LIN {X 0,Y 355.23,Z 732.233,A -85,B 0,C 180,E1 -13592.268,E2 -13592.268} C_VEL
LIN {X 0,Y 355.091,Z 732.252,A -85,B 0,C 180,E1 -13596.82,E2 -13596.82} C_VEL
LIN {X 0,Y 354.959,Z 732.267,A -85,B 0,C 180,E1 -13600.265,E2 -13600.265} C_VEL
LIN {X 0,Y 354.946,Z 732.27,A -85,B 0,C 180,E1 -13604.019,E2 -13604.019} C_VEL
LIN {X 0,Y 354.926,Z 732.273,A -85,B 0,C 180,E1 -13608.108,E2 -13608.108} C_VEL
LIN {X 0,Y 354.811,Z 732.288,A -85,B 0,C 180,E1 -13612.108,E2 -13612.108} C_VEL
LIN {X 0,Y 354.852,Z 732.28,A -85,B 0,C 180,E1 -13614.577,E2 -13614.577} C_VEL
LIN {X 0,Y 354.804,Z 732.288,A -85,B 0,C 180,E1 -13618.385,E2 -13618.385} C_VEL
LIN {X 0,Y 354.79,Z 732.291,A -85,B 0,C 180,E1 -13622.333,E2 -13622.333} C_VEL
LIN {X 0,Y 354.825,Z 732.285,A -85,B 0,C 180,E1 -13625.699,E2 -13625.699} C_VEL
LIN {X 0,Y 354.827,Z 732.283,A -85,B 0,C 180,E1 -13629.424,E2 -13629.424} C_VEL
LIN {X 0,Y 354.837,Z 732.433,A -85,B 0,C 180,E1 -13633.462,E2 -13633.462} C_VEL
LIN {X 0,Y 358.442,Z 744.759,A -85,B 0,C 180,E1 -13634.507,E2 -13634.507} C_VEL
LIN {X 0,Y 360.272,Z 752.132,A -85,B 0,C 180,E1 -13635.248,E2 -13635.248} C_VEL
LIN {X 0,Y 359.509,Z 762.827,A -85,B 0,C 180,E1 -13636.329,E2 -13636.329} C_VEL
LIN {X 0,Y 358.79,Z 772.72,A -85,B 0,C 180,E1 -13637.56,E2 -13637.56} C_VEL
LIN {X 0,Y 358.14,Z 780.809,A -85,B 0,C 180,E1 -13638.776,E2 -13638.776} C_VEL
LIN {X 0,Y 357.07,Z 784.926,A -85,B 0,C 180,E1 -13639.442,E2 -13639.442} C_VEL
LIN {X 0,Y 353.693,Z 791.298,A -85,B 0,C 180,E1 -13640.535,E2 -13640.535} C_VEL
LIN {X 0,Y 350.384,Z 797.153,A -85,B 0,C 180,E1 -13641.719,E2 -13641.719} C_VEL
LIN {X 0,Y 349.435,Z 800.343,A -85,B 0,C 180,E1 -13642.517,E2 -13642.517} C_VEL
LIN {X 0,Y 348.883,Z 806.047,A -85,B 0,C 180,E1 -13644.254,E2 -13644.254} C_VEL
LIN {X 0,Y 348.465,Z 811.428,A -85,B 0,C 180,E1 -13646.383,E2 -13646.383} C_VEL
LIN {X 0,Y 348.168,Z 814.944,A -85,B 0,C 180,E1 -13648.343,E2 -13648.343} C_VEL
LIN {X 0,Y 348.021,Z 817.216,A -85,B 0,C 180,E1 -13650.268,E2 -13650.268} C_VEL
LIN {X 0,Y 348.097,Z 818.5,A -85,B 0,C 180,E1 -13652.667,E2 -13652.667} C_VEL
LIN {X 0,Y 348.403,Z 818.075,A -85,B 0,C 180,E1 -13654.937,E2 -13654.937} C_VEL
LIN {X 0,Y 348.678,Z 817.181,A -85,B 0,C 180,E1 -13656.226,E2 -13656.226} C_VEL
LIN {X 0,Y 349.127,Z 815.318,A -85,B 0,C 180,E1 -13657.819,E2 -13657.819} C_VEL
LIN {X 0,Y 349.648,Z 812.667,A -85,B 0,C 180,E1 -13659.405,E2 -13659.405} C_VEL
LIN {X 0,Y 350.447,Z 808.387,A -85,B 0,C 180,E1 -13661.284,E2 -13661.284} C_VEL
LIN {X 0,Y 351.444,Z 802.773,A -85,B 0,C 180,E1 -13663.145,E2 -13663.145} C_VEL
LIN {X 0,Y 352.623,Z 795.572,A -85,B 0,C 180,E1 -13664.983,E2 -13664.983} C_VEL
LIN {X 0,Y 353.849,Z 787.076,A -85,B 0,C 180,E1 -13666.711,E2 -13666.711} C_VEL
LIN {X 0,Y 355.031,Z 778.224,A -85,B 0,C 180,E1 -13668.148,E2 -13668.148} C_VEL
LIN {X 0,Y 356.154,Z 768.152,A -85,B 0,C 180,E1 -13669.483,E2 -13669.483} C_VEL
LIN {X 0,Y 356.951,Z 758.725,A -85,B 0,C 180,E1 -13670.508,E2 -13670.508} C_VEL
LIN {X 0,Y 354.065,Z 748.897,A -85,B 0,C 180,E1 -13671.697,E2 -13671.697} C_VEL
LIN {X 0,Y 350.313,Z 738.899,A -85,B 0,C 180,E1 -13672.797,E2 -13672.797} C_VEL
LIN {X 0,Y 348.038,Z 733.135,A -85,B 0,C 180,E1 -13673.405,E2 -13673.405} C_VEL
LIN {X 0,Y 348.206,Z 733.113,A -85,B 0,C 180,E1 -13677.686,E2 -13677.686} C_VEL
LIN {X 0,Y 348.307,Z 733.1,A -85,B 0,C 180,E1 -13680,E2 -13680} C_VEL
LIN {X 0,Y 348.206,Z 733.106,A -85,B 0,C 180,E1 -13682.313,E2 -13682.313} C_VEL
LIN {X 0,Y 348.091,Z 733.123,A -85,B 0,C 180,E1 -13686.958,E2 -13686.958} C_VEL
LIN {X 0,Y 347.931,Z 733.145,A -85,B 0,C 180,E1 -13690.474,E2 -13690.474} C_VEL
LIN {X 0,Y 347.902,Z 733.146,A -85,B 0,C 180,E1 -13694.15,E2 -13694.15} C_VEL
LIN {X 0,Y 347.894,Z 733.145,A -85,B 0,C 180,E1 -13698.29,E2 -13698.29} C_VEL
LIN {X 0,Y 347.77,Z 733.16,A -85,B 0,C 180,E1 -13701.626,E2 -13701.626} C_VEL
LIN {X 0,Y 347.814,Z 733.16,A -85,B 0,C 180,E1 -13705.108,E2 -13705.108} C_VEL
LIN {X 0,Y 347.811,Z 733.161,A -85,B 0,C 180,E1 -13707.694,E2 -13707.694} C_VEL
LIN {X 0,Y 347.752,Z 733.168,A -85,B 0,C 180,E1 -13710.348,E2 -13710.348} C_VEL
LIN {X 0,Y 347.751,Z 733.169,A -85,B 0,C 180,E1 -13714.044,E2 -13714.044} C_VEL
LIN {X 0,Y 347.764,Z 733.169,A -85,B 0,C 180,E1 -13717.321,E2 -13717.321} C_VEL
LIN {X 0,Y 347.757,Z 733.181,A -85,B 0,C 180,E1 -13720.819,E2 -13720.819} C_VEL
LIN {X 0,Y 348.955,Z 738.713,A -85,B 0,C 180,E1 -13724.033,E2 -13724.033} C_VEL
LIN {X 0,Y 350.122,Z 744.422,A -85,B 0,C 180,E1 -13726.962,E2 -13726.962} C_VEL
LIN {X 0,Y 351.537,Z 751.508,A -85,B 0,C 180,E1 -13730.226,E2 -13730.226} C_VEL
LIN {X 0,Y 352.141,Z 756.915,A -85,B 0,C 180,E1 -13732.473,E2 -13732.473} C_VEL
LIN {X 0,Y 350.934,Z 766.228,A -85,B 0,C 180,E1 -13735.892,E2 -13735.892} C_VEL
LIN {X 0,Y 349.45,Z 779.49,A -85,B 0,C 180,E1 -13740.479,E2 -13740.479} C_VEL
LIN {X 0,Y 348.465,Z 791.054,A -85,B 0,C 180,E1 -13744.302,E2 -13744.302} C_VEL
LIN {X 0,Y 347.758,Z 802.825,A -85,B 0,C 180,E1 -13748.058,E2 -13748.058} C_VEL
LIN {X 0,Y 350.244,Z 818.097,A -85,B 0,C 180,E1 -13748.869,E2 -13748.869} C_VEL
LIN {X 0,Y 351.372,Z 830.122,A -85,B 0,C 180,E1 -13749.648,E2 -13749.648} C_VEL
LIN {X 0,Y 351.672,Z 841.978,A -85,B 0,C 180,E1 -13750.557,E2 -13750.557} C_VEL
LIN {X 0,Y 351.564,Z 853.712,A -85,B 0,C 180,E1 -13751.648,E2 -13751.648} C_VEL
LIN {X 0,Y 351.503,Z 860.57,A -85,B 0,C 180,E1 -13752.397,E2 -13752.397} C_VEL
LIN {X 0,Y 350.096,Z 871.051,A -85,B 0,C 180,E1 -13753.677,E2 -13753.677} C_VEL
LIN {X 0,Y 348.932,Z 881.081,A -85,B 0,C 180,E1 -13755.193,E2 -13755.193} C_VEL
LIN {X 0,Y 347.998,Z 890.121,A -85,B 0,C 180,E1 -13756.868,E2 -13756.868} C_VEL
LIN {X 0,Y 347.338,Z 897.875,A -85,B 0,C 180,E1 -13758.622,E2 -13758.622} C_VEL
LIN {X 0,Y 346.927,Z 905.128,A -85,B 0,C 180,E1 -13760.673,E2 -13760.673} C_VEL
LIN {X 0,Y 346.843,Z 910.019,A -85,B 0,C 180,E1 -13762.432,E2 -13762.432} C_VEL
LIN {X 0,Y 346.898,Z 913.8,A -85,B 0,C 180,E1 -13764.186,E2 -13764.186} C_VEL
LIN {X 0,Y 347.05,Z 915.739,A -85,B 0,C 180,E1 -13765.354,E2 -13765.354} C_VEL
LIN {X 0,Y 347.128,Z 917.246,A -85,B 0,C 180,E1 -13766.518,E2 -13766.518} C_VEL
LIN {X 0,Y 347.158,Z 918.314,A -85,B 0,C 180,E1 -13767.679,E2 -13767.679} C_VEL
LIN {X 0,Y 347.23,Z 918.922,A -85,B 0,C 180,E1 -13768.84,E2 -13768.84} C_VEL
LIN {X 0,Y 347.29,Z 919.114,A -85,B 0,C 180,E1 -13770,E2 -13770} C_VEL
LIN {X 0,Y 347.241,Z 918.877,A -85,B 0,C 180,E1 -13771.16,E2 -13771.16} C_VEL
LIN {X 0,Y 347.186,Z 918.212,A -85,B 0,C 180,E1 -13772.32,E2 -13772.32} C_VEL
LIN {X 0,Y 347.148,Z 917.076,A -85,B 0,C 180,E1 -13773.482,E2 -13773.482} C_VEL
LIN {X 0,Y 347.021,Z 914.544,A -85,B 0,C 180,E1 -13775.229,E2 -13775.229} C_VEL
LIN {X 0,Y 346.945,Z 910.936,A -85,B 0,C 180,E1 -13776.981,E2 -13776.981} C_VEL
LIN {X 0,Y 346.942,Z 906.157,A -85,B 0,C 180,E1 -13778.739,E2 -13778.739} C_VEL
LIN {X 0,Y 347.233,Z 898.965,A -85,B 0,C 180,E1 -13780.791,E2 -13780.791} C_VEL
LIN {X 0,Y 347.794,Z 891.13,A -85,B 0,C 180,E1 -13782.546,E2 -13782.546} C_VEL
LIN {X 0,Y 348.508,Z 883.149,A -85,B 0,C 180,E1 -13784.004,E2 -13784.004} C_VEL
LIN {X 0,Y 349.435,Z 873.459,A -85,B 0,C 180,E1 -13785.455,E2 -13785.455} C_VEL
LIN {X 0,Y 350.509,Z 862.791,A -85,B 0,C 180,E1 -13786.752,E2 -13786.752} C_VEL
LIN {X 0,Y 351.002,Z 857.17,A -85,B 0,C 180,E1 -13787.328,E2 -13787.328} C_VEL
LIN {X 0,Y 350.463,Z 844.972,A -85,B 0,C 180,E1 -13788.412,E2 -13788.412} C_VEL
LIN {X 0,Y 349.684,Z 831.983,A -85,B 0,C 180,E1 -13789.319,E2 -13789.319} C_VEL
LIN {X 0,Y 348.451,Z 818.444,A -85,B 0,C 180,E1 -13790.02,E2 -13790.02} C_VEL
LIN {X 0,Y 347.553,Z 809.771,A -85,B 0,C 180,E1 -13790.376,E2 -13790.376} C_VEL
LIN {X 0,Y 348.209,Z 799.166,A -85,B 0,C 180,E1 -13793.808,E2 -13793.808} C_VEL
LIN {X 0,Y 349.199,Z 787.298,A -85,B 0,C 180,E1 -13797.681,E2 -13797.681} C_VEL
LIN {X 0,Y 350.29,Z 775.966,A -85,B 0,C 180,E1 -13801.443,E2 -13801.443} C_VEL
LIN {X 0,Y 351.553,Z 765.595,A -85,B 0,C 180,E1 -13804.951,E2 -13804.951} C_VEL
LIN {X 0,Y 352.474,Z 758.03,A -85,B 0,C 180,E1 -13807.561,E2 -13807.561} C_VEL
LIN {X 0,Y 351.825,Z 753.478,A -85,B 0,C 180,E1 -13809.252,E2 -13809.252} C_VEL
LIN {X 0,Y 350.11,Z 744.683,A -85,B 0,C 180,E1 -13812.661,E2 -13812.661} C_VEL
LIN {X 0,Y 348.125,Z 735.001,A -85,B 0,C 180,E1 -13816.654,E2 -13816.654} C_VEL
LIN {X 0,Y 347.747,Z 733.17,A -85,B 0,C 180,E1 -13817.486,E2 -13817.486} C_VEL
LIN {X 0,Y 347.753,Z 733.168,A -85,B 0,C 180,E1 -13821.207,E2 -13821.207} C_VEL
LIN {X 0,Y 347.79,Z 733.161,A -85,B 0,C 180,E1 -13824.125,E2 -13824.125} C_VEL
LIN {X 0,Y 347.74,Z 733.169,A -85,B 0,C 180,E1 -13828.086,E2 -13828.086} C_VEL
LIN {X 0,Y 347.806,Z 733.157,A -85,B 0,C 180,E1 -13830.99,E2 -13830.99} C_VEL
LIN {X 0,Y 347.833,Z 733.157,A -85,B 0,C 180,E1 -13833.608,E2 -13833.608} C_VEL
LIN {X 0,Y 347.787,Z 733.164,A -85,B 0,C 180,E1 -13836.162,E2 -13836.162} C_VEL
LIN {X 0,Y 347.813,Z 733.161,A -85,B 0,C 180,E1 -13839.909,E2 -13839.909} C_VEL
LIN {X 0,Y 347.868,Z 733.154,A -85,B 0,C 180,E1 -13842.359,E2 -13842.359} C_VEL
LIN {X 0,Y 347.899,Z 733.149,A -85,B 0,C 180,E1 -13845.971,E2 -13845.971} C_VEL
LIN {X 0,Y 347.93,Z 733.142,A -85,B 0,C 180,E1 -13849.526,E2 -13849.526} C_VEL
LIN {X 0,Y 348.093,Z 733.123,A -85,B 0,C 180,E1 -13853.042,E2 -13853.042} C_VEL
LIN {X 0,Y 348.197,Z 733.109,A -85,B 0,C 180,E1 -13857.687,E2 -13857.687} C_VEL
LIN {X 0,Y 348.305,Z 733.096,A -85,B 0,C 180,E1 -13860,E2 -13860} C_VEL
LIN {X 0,Y 348.205,Z 733.11,A -85,B 0,C 180,E1 -13862.314,E2 -13862.314} C_VEL
LIN {X 0,Y 348.069,Z 733.13,A -85,B 0,C 180,E1 -13866.959,E2 -13866.959} C_VEL
LIN {X 0,Y 347.899,Z 733.148,A -85,B 0,C 180,E1 -13870.475,E2 -13870.475} C_VEL
LIN {X 0,Y 347.9,Z 733.146,A -85,B 0,C 180,E1 -13874.15,E2 -13874.15} C_VEL
LIN {X 0,Y 347.831,Z 733.155,A -85,B 0,C 180,E1 -13878.259,E2 -13878.259} C_VEL
LIN {X 0,Y 347.766,Z 733.166,A -85,B 0,C 180,E1 -13881.625,E2 -13881.625} C_VEL
LIN {X 0,Y 347.741,Z 733.17,A -85,B 0,C 180,E1 -13885.114,E2 -13885.114} C_VEL
LIN {X 0,Y 347.739,Z 733.17,A -85,B 0,C 180,E1 -13887.7,E2 -13887.7} C_VEL
LIN {X 0,Y 347.742,Z 733.166,A -85,B 0,C 180,E1 -13890.349,E2 -13890.349} C_VEL
LIN {X 0,Y 347.749,Z 733.167,A -85,B 0,C 180,E1 -13894.044,E2 -13894.044} C_VEL
LIN {X 0,Y 347.756,Z 733.167,A -85,B 0,C 180,E1 -13897.322,E2 -13897.322} C_VEL
LIN {X 0,Y 347.741,Z 733.17,A -85,B 0,C 180,E1 -13901.601,E2 -13901.601} C_VEL
LIN {X 0,Y 347.701,Z 733.171,A -85,B 0,C 180,E1 -13905.028,E2 -13905.028} C_VEL
LIN {X 0,Y 347.741,Z 733.169,A -85,B 0,C 180,E1 -13908.4,E2 -13908.4} C_VEL
LIN {X 0,Y 347.763,Z 733.168,A -85,B 0,C 180,E1 -13912.014,E2 -13912.014} C_VEL
LIN {X 0,Y 347.744,Z 733.166,A -85,B 0,C 180,E1 -13915.536,E2 -13915.536} C_VEL
LIN {X 0,Y 347.746,Z 733.17,A -85,B 0,C 180,E1 -13918.3,E2 -13918.3} C_VEL
LIN {X 0,Y 347.745,Z 733.166,A -85,B 0,C 180,E1 -13920.985,E2 -13920.985} C_VEL
LIN {X 0,Y 347.735,Z 733.167,A -85,B 0,C 180,E1 -13923.6,E2 -13923.6} C_VEL
LIN {X 0,Y 347.751,Z 733.168,A -85,B 0,C 180,E1 -13926.159,E2 -13926.159} C_VEL
LIN {X 0,Y 347.808,Z 733.158,A -85,B 0,C 180,E1 -13929.909,E2 -13929.909} C_VEL
LIN {X 0,Y 347.834,Z 733.154,A -85,B 0,C 180,E1 -13933.568,E2 -13933.568} C_VEL
LIN {X 0,Y 347.889,Z 733.15,A -85,B 0,C 180,E1 -13937.161,E2 -13937.161} C_VEL
LIN {X 0,Y 347.936,Z 733.146,A -85,B 0,C 180,E1 -13940.701,E2 -13940.701} C_VEL
LIN {X 0,Y 348.039,Z 733.129,A -85,B 0,C 180,E1 -13944.205,E2 -13944.205} C_VEL
LIN {X 0,Y 348.19,Z 733.111,A -85,B 0,C 180,E1 -13947.687,E2 -13947.687} C_VEL
LIN {X 0,Y 348.119,Z 733.124,A -85,B 0,C 180,E1 -13951.157,E2 -13951.157} C_VEL
LIN {X 0,Y 348.192,Z 733.11,A -85,B 0,C 180,E1 -13952.314,E2 -13952.314} C_VEL
LIN {X 0,Y 348.058,Z 733.129,A -85,B 0,C 180,E1 -13956.959,E2 -13956.959} C_VEL
LIN {X 0,Y 347.899,Z 733.146,A -85,B 0,C 180,E1 -13960.475,E2 -13960.475} C_VEL
LIN {X 0,Y 347.902,Z 733.147,A -85,B 0,C 180,E1 -13964.15,E2 -13964.15} C_VEL
LIN {X 0,Y 347.894,Z 733.147,A -85,B 0,C 180,E1 -13968.29,E2 -13968.29} C_VEL
LIN {X 0,Y 347.768,Z 733.167,A -85,B 0,C 180,E1 -13971.625,E2 -13971.625} C_VEL
LIN {X 0,Y 347.772,Z 733.162,A -85,B 0,C 180,E1 -13975.112,E2 -13975.112} C_VEL
LIN {X 0,Y 347.741,Z 733.169,A -85,B 0,C 180,E1 -13977.7,E2 -13977.7} C_VEL
LIN {X 0,Y 347.744,Z 733.168,A -85,B 0,C 180,E1 -13980.349,E2 -13980.349} C_VEL
LIN {X 0,Y 347.751,Z 733.169,A -85,B 0,C 180,E1 -13984.044,E2 -13984.044} C_VEL
LIN {X 0,Y 347.764,Z 733.162,A -85,B 0,C 180,E1 -13987.321,E2 -13987.321} C_VEL
LIN {X 0,Y 347.736,Z 733.172,A -85,B 0,C 180,E1 -13990.297,E2 -13990.297} C_VEL
LIN {X 0,Y 347.768,Z 733.163,A -85,B 0,C 180,E1 -13993.143,E2 -13993.143} C_VEL
LIN {X 0,Y 351.234,Z 745.101,A -85,B 0,C 180,E1 -13994.174,E2 -13994.174} C_VEL
LIN {X 0,Y 353.253,Z 752.532,A -85,B 0,C 180,E1 -13994.933,E2 -13994.933} C_VEL
LIN {X 0,Y 352.761,Z 762.272,A -85,B 0,C 180,E1 -13995.928,E2 -13995.928} C_VEL
LIN {X 0,Y 351.956,Z 772.866,A -85,B 0,C 180,E1 -13997.24,E2 -13997.24} C_VEL
LIN {X 0,Y 351.147,Z 782.229,A -85,B 0,C 180,E1 -13998.663,E2 -13998.663} C_VEL
LIN {X 0,Y 350.27,Z 791.601,A -85,B 0,C 180,E1 -14000.427,E2 -14000.427} C_VEL
LIN {X 0,Y 349.541,Z 799.315,A -85,B 0,C 180,E1 -14002.234,E2 -14002.234} C_VEL
LIN {X 0,Y 349.435,Z 800.343,A -85,B 0,C 180,E1 -14002.517,E2 -14002.517} C_VEL
LIN {X 0,Y 348.513,Z 803.347,A -85,B 0,C 180,E1 -14003.34,E2 -14003.34} C_VEL
LIN {X 0,Y 345.338,Z 807.953,A -85,B 0,C 180,E1 -14004.691,E2 -14004.691} C_VEL
LIN {X 0,Y 342.198,Z 811.889,A -85,B 0,C 180,E1 -14006.117,E2 -14006.117} C_VEL
LIN {X 0,Y 341.352,Z 813.811,A -85,B 0,C 180,E1 -14007.044,E2 -14007.044} C_VEL
LIN {X 0,Y 341.084,Z 816.896,A -85,B 0,C 180,E1 -14008.994,E2 -14008.994} C_VEL
LIN {X 0,Y 340.994,Z 818.317,A -85,B 0,C 180,E1 -14010.353,E2 -14010.353} C_VEL
LIN {X 0,Y 341.074,Z 819.469,A -85,B 0,C 180,E1 -14012.38,E2 -14012.38} C_VEL
LIN {X 0,Y 341.392,Z 819.241,A -85,B 0,C 180,E1 -14014.932,E2 -14014.932} C_VEL
LIN {X 0,Y 341.892,Z 817.661,A -85,B 0,C 180,E1 -14017.01,E2 -14017.01} C_VEL
LIN {X 0,Y 342.544,Z 815.006,A -85,B 0,C 180,E1 -14018.958,E2 -14018.958} C_VEL
LIN {X 0,Y 343.28,Z 811.201,A -85,B 0,C 180,E1 -14020.878,E2 -14020.878} C_VEL
LIN {X 0,Y 344.294,Z 806.037,A -85,B 0,C 180,E1 -14022.783,E2 -14022.783} C_VEL
LIN {X 0,Y 345.475,Z 799.43,A -85,B 0,C 180,E1 -14024.665,E2 -14024.665} C_VEL
LIN {X 0,Y 346.688,Z 792.011,A -85,B 0,C 180,E1 -14026.355,E2 -14026.355} C_VEL
LIN {X 0,Y 347.787,Z 784.502,A -85,B 0,C 180,E1 -14027.75,E2 -14027.75} C_VEL
LIN {X 0,Y 349.124,Z 774.386,A -85,B 0,C 180,E1 -14029.268,E2 -14029.268} C_VEL
LIN {X 0,Y 350.266,Z 763.595,A -85,B 0,C 180,E1 -14030.574,E2 -14030.574} C_VEL
LIN {X 0,Y 350.35,Z 760.277,A -85,B 0,C 180,E1 -14030.936,E2 -14030.936} C_VEL
LIN {X 0,Y 347.237,Z 749.774,A -85,B 0,C 180,E1 -14032.256,E2 -14032.256} C_VEL
LIN {X 0,Y 343.468,Z 739.901,A -85,B 0,C 180,E1 -14033.391,E2 -14033.391} C_VEL
LIN {X 0,Y 341.173,Z 734.849,A -85,B 0,C 180,E1 -14033.94,E2 -14033.94} C_VEL
LIN {X 0,Y 341.017,Z 734.004,A -85,B 0,C 180,E1 -14034.011,E2 -14034.011} C_VEL
LIN {X 0,Y 341.168,Z 733.989,A -85,B 0,C 180,E1 -14037.639,E2 -14037.639} C_VEL
LIN {X 0,Y 341.258,Z 733.978,A -85,B 0,C 180,E1 -14040,E2 -14040} C_VEL
LIN {X 0,Y 341.168,Z 733.982,A -85,B 0,C 180,E1 -14042.361,E2 -14042.361} C_VEL
LIN {X 0,Y 341.06,Z 733.999,A -85,B 0,C 180,E1 -14047.102,E2 -14047.102} C_VEL
LIN {X 0,Y 340.874,Z 734.023,A -85,B 0,C 180,E1 -14050.694,E2 -14050.694} C_VEL
LIN {X 0,Y 340.866,Z 734.021,A -85,B 0,C 180,E1 -14054.325,E2 -14054.325} C_VEL
LIN {X 0,Y 340.84,Z 734.024,A -85,B 0,C 180,E1 -14058.466,E2 -14058.466} C_VEL
LIN {X 0,Y 340.72,Z 734.039,A -85,B 0,C 180,E1 -14061.841,E2 -14061.841} C_VEL
LIN {X 0,Y 340.775,Z 734.037,A -85,B 0,C 180,E1 -14065.664,E2 -14065.664} C_VEL
LIN {X 0,Y 340.731,Z 734.04,A -85,B 0,C 180,E1 -14068.321,E2 -14068.321} C_VEL
LIN {X 0,Y 340.7,Z 734.043,A -85,B 0,C 180,E1 -14071.044,E2 -14071.044} C_VEL
LIN {X 0,Y 340.721,Z 734.043,A -85,B 0,C 180,E1 -14075.279,E2 -14075.279} C_VEL
LIN {X 0,Y 340.712,Z 734.049,A -85,B 0,C 180,E1 -14078.386,E2 -14078.386} C_VEL
LIN {X 0,Y 340.724,Z 734.107,A -85,B 0,C 180,E1 -14080.01,E2 -14080.01} C_VEL
LIN {X 0,Y 341.924,Z 739.628,A -85,B 0,C 180,E1 -14083.391,E2 -14083.391} C_VEL
LIN {X 0,Y 343.155,Z 745.722,A -85,B 0,C 180,E1 -14086.64,E2 -14086.64} C_VEL
LIN {X 0,Y 344.587,Z 752.85,A -85,B 0,C 180,E1 -14090.025,E2 -14090.025} C_VEL
LIN {X 0,Y 345.148,Z 756.489,A -85,B 0,C 180,E1 -14091.607,E2 -14091.607} C_VEL
LIN {X 0,Y 345.136,Z 758.878,A -85,B 0,C 180,E1 -14092.576,E2 -14092.576} C_VEL
LIN {X 0,Y 343.943,Z 767.473,A -85,B 0,C 180,E1 -14095.811,E2 -14095.811} C_VEL
LIN {X 0,Y 342.385,Z 780.646,A -85,B 0,C 180,E1 -14100.486,E2 -14100.486} C_VEL
LIN {X 0,Y 341.397,Z 792.174,A -85,B 0,C 180,E1 -14104.386,E2 -14104.386} C_VEL
LIN {X 0,Y 340.78,Z 801.684,A -85,B 0,C 180,E1 -14107.439,E2 -14107.439} C_VEL
LIN {X 0,Y 343.371,Z 816.716,A -85,B 0,C 180,E1 -14108.293,E2 -14108.293} C_VEL
LIN {X 0,Y 344.673,Z 829.763,A -85,B 0,C 180,E1 -14109.173,E2 -14109.173} C_VEL
LIN {X 0,Y 344.926,Z 842.378,A -85,B 0,C 180,E1 -14110.191,E2 -14110.191} C_VEL
LIN {X 0,Y 344.69,Z 854.862,A -85,B 0,C 180,E1 -14111.422,E2 -14111.422} C_VEL
LIN {X 0,Y 344.566,Z 861.431,A -85,B 0,C 180,E1 -14112.184,E2 -14112.184} C_VEL
LIN {X 0,Y 342.986,Z 872.499,A -85,B 0,C 180,E1 -14113.635,E2 -14113.635} C_VEL
LIN {X 0,Y 341.896,Z 881.316,A -85,B 0,C 180,E1 -14115.046,E2 -14115.046} C_VEL
LIN {X 0,Y 341.048,Z 889.379,A -85,B 0,C 180,E1 -14116.595,E2 -14116.595} C_VEL
LIN {X 0,Y 340.315,Z 897.076,A -85,B 0,C 180,E1 -14118.384,E2 -14118.384} C_VEL
LIN {X 0,Y 339.975,Z 902.361,A -85,B 0,C 180,E1 -14119.88,E2 -14119.88} C_VEL
LIN {X 0,Y 339.773,Z 907.59,A -85,B 0,C 180,E1 -14121.675,E2 -14121.675} C_VEL
LIN {X 0,Y 339.801,Z 910.959,A -85,B 0,C 180,E1 -14123.107,E2 -14123.107} C_VEL
LIN {X 0,Y 339.992,Z 914.762,A -85,B 0,C 180,E1 -14125.257,E2 -14125.257} C_VEL
LIN {X 0,Y 340.085,Z 916.259,A -85,B 0,C 180,E1 -14126.445,E2 -14126.445} C_VEL
LIN {X 0,Y 340.118,Z 917.295,A -85,B 0,C 180,E1 -14127.631,E2 -14127.631} C_VEL
LIN {X 0,Y 340.198,Z 917.888,A -85,B 0,C 180,E1 -14128.816,E2 -14128.816} C_VEL
LIN {X 0,Y 340.266,Z 918.068,A -85,B 0,C 180,E1 -14130,E2 -14130} C_VEL
LIN {X 0,Y 340.213,Z 917.818,A -85,B 0,C 180,E1 -14131.184,E2 -14131.184} C_VEL
LIN {X 0,Y 340.156,Z 917.115,A -85,B 0,C 180,E1 -14132.368,E2 -14132.368} C_VEL
LIN {X 0,Y 340.106,Z 915.956,A -85,B 0,C 180,E1 -14133.554,E2 -14133.554} C_VEL
LIN {X 0,Y 339.971,Z 913.383,A -85,B 0,C 180,E1 -14135.338,E2 -14135.338} C_VEL
LIN {X 0,Y 339.88,Z 909.726,A -85,B 0,C 180,E1 -14137.127,E2 -14137.127} C_VEL
LIN {X 0,Y 339.911,Z 904.901,A -85,B 0,C 180,E1 -14138.921,E2 -14138.921} C_VEL
LIN {X 0,Y 340.157,Z 898.783,A -85,B 0,C 180,E1 -14140.716,E2 -14140.716} C_VEL
LIN {X 0,Y 340.688,Z 891.179,A -85,B 0,C 180,E1 -14142.51,E2 -14142.51} C_VEL
LIN {X 0,Y 341.425,Z 883.438,A -85,B 0,C 180,E1 -14143.997,E2 -14143.997} C_VEL
LIN {X 0,Y 342.318,Z 874.012,A -85,B 0,C 180,E1 -14145.48,E2 -14145.48} C_VEL
LIN {X 0,Y 343.409,Z 863.657,A -85,B 0,C 180,E1 -14146.802,E2 -14146.802} C_VEL
LIN {X 0,Y 343.936,Z 856.845,A -85,B 0,C 180,E1 -14147.542,E2 -14147.542} C_VEL
LIN {X 0,Y 343.448,Z 844.854,A -85,B 0,C 180,E1 -14148.647,E2 -14148.647} C_VEL
LIN {X 0,Y 342.636,Z 831.043,A -85,B 0,C 180,E1 -14149.644,E2 -14149.644} C_VEL
LIN {X 0,Y 341.455,Z 817.895,A -85,B 0,C 180,E1 -14150.347,E2 -14150.347} C_VEL
LIN {X 0,Y 340.567,Z 808.849,A -85,B 0,C 180,E1 -14150.735,E2 -14150.735} C_VEL
LIN {X 0,Y 341.336,Z 796.876,A -85,B 0,C 180,E1 -14154.701,E2 -14154.701} C_VEL
LIN {X 0,Y 342.271,Z 786.494,A -85,B 0,C 180,E1 -14158.182,E2 -14158.182} C_VEL
LIN {X 0,Y 343.46,Z 774.864,A -85,B 0,C 180,E1 -14162.142,E2 -14162.142} C_VEL
LIN {X 0,Y 344.788,Z 764.543,A -85,B 0,C 180,E1 -14165.725,E2 -14165.725} C_VEL
LIN {X 0,Y 345.481,Z 759.219,A -85,B 0,C 180,E1 -14167.61,E2 -14167.61} C_VEL
LIN {X 0,Y 344.878,Z 754.873,A -85,B 0,C 180,E1 -14169.252,E2 -14169.252} C_VEL
LIN {X 0,Y 343.25,Z 746.62,A -85,B 0,C 180,E1 -14172.515,E2 -14172.515} C_VEL
LIN {X 0,Y 341.502,Z 738.052,A -85,B 0,C 180,E1 -14176.078,E2 -14176.078} C_VEL
LIN {X 0,Y 340.733,Z 734.042,A -85,B 0,C 180,E1 -14177.816,E2 -14177.816} C_VEL
LIN {X 0,Y 340.734,Z 734.043,A -85,B 0,C 180,E1 -14181.773,E2 -14181.773} C_VEL
LIN {X 0,Y 340.724,Z 734.044,A -85,B 0,C 180,E1 -14185.595,E2 -14185.595} C_VEL
LIN {X 0,Y 340.705,Z 734.042,A -85,B 0,C 180,E1 -14188.956,E2 -14188.956} C_VEL
LIN {X 0,Y 340.78,Z 734.034,A -85,B 0,C 180,E1 -14192.474,E2 -14192.474} C_VEL
LIN {X 0,Y 340.756,Z 734.038,A -85,B 0,C 180,E1 -14195.638,E2 -14195.638} C_VEL
LIN {X 0,Y 340.741,Z 734.038,A -85,B 0,C 180,E1 -14199.474,E2 -14199.474} C_VEL
LIN {X 0,Y 340.86,Z 734.027,A -85,B 0,C 180,E1 -14201.984,E2 -14201.984} C_VEL
LIN {X 0,Y 340.871,Z 734.022,A -85,B 0,C 180,E1 -14205.705,E2 -14205.705} C_VEL
LIN {X 0,Y 340.873,Z 734.021,A -85,B 0,C 180,E1 -14209.306,E2 -14209.306} C_VEL
LIN {X 0,Y 341.061,Z 734,A -85,B 0,C 180,E1 -14212.898,E2 -14212.898} C_VEL
LIN {X 0,Y 341.159,Z 733.985,A -85,B 0,C 180,E1 -14217.639,E2 -14217.639} C_VEL
LIN {X 0,Y 341.256,Z 733.974,A -85,B 0,C 180,E1 -14220,E2 -14220} C_VEL
LIN {X 0,Y 341.166,Z 733.987,A -85,B 0,C 180,E1 -14222.361,E2 -14222.361} C_VEL
LIN {X 0,Y 341.018,Z 734.007,A -85,B 0,C 180,E1 -14227.103,E2 -14227.103} C_VEL
LIN {X 0,Y 340.85,Z 734.028,A -85,B 0,C 180,E1 -14230.695,E2 -14230.695} C_VEL
LIN {X 0,Y 340.865,Z 734.023,A -85,B 0,C 180,E1 -14234.325,E2 -14234.325} C_VEL
LIN {X 0,Y 340.788,Z 734.032,A -85,B 0,C 180,E1 -14238.441,E2 -14238.441} C_VEL
LIN {X 0,Y 340.719,Z 734.042,A -85,B 0,C 180,E1 -14241.842,E2 -14241.842} C_VEL
LIN {X 0,Y 340.678,Z 734.049,A -85,B 0,C 180,E1 -14245.672,E2 -14245.672} C_VEL
LIN {X 0,Y 340.685,Z 734.045,A -85,B 0,C 180,E1 -14248.325,E2 -14248.325} C_VEL
LIN {X 0,Y 340.696,Z 734.045,A -85,B 0,C 180,E1 -14251.045,E2 -14251.045} C_VEL
LIN {X 0,Y 340.717,Z 734.043,A -85,B 0,C 180,E1 -14255.279,E2 -14255.279} C_VEL
LIN {X 0,Y 340.694,Z 734.044,A -85,B 0,C 180,E1 -14258.382,E2 -14258.382} C_VEL
LIN {X 0,Y 340.693,Z 734.048,A -85,B 0,C 180,E1 -14262.044,E2 -14262.044} C_VEL
LIN {X 0,Y 340.651,Z 734.052,A -85,B 0,C 180,E1 -14266.228,E2 -14266.228} C_VEL
LIN {X 0,Y 340.67,Z 734.047,A -85,B 0,C 180,E1 -14268.688,E2 -14268.688} C_VEL
LIN {X 0,Y 340.72,Z 734.043,A -85,B 0,C 180,E1 -14271.771,E2 -14271.771} C_VEL
LIN {X 0,Y 340.723,Z 734.041,A -85,B 0,C 180,E1 -14275.596,E2 -14275.596} C_VEL
LIN {X 0,Y 340.694,Z 734.044,A -85,B 0,C 180,E1 -14278.955,E2 -14278.955} C_VEL
LIN {X 0,Y 340.711,Z 734.042,A -85,B 0,C 180,E1 -14283.012,E2 -14283.012} C_VEL
LIN {X 0,Y 340.703,Z 734.045,A -85,B 0,C 180,E1 -14286.925,E2 -14286.925} C_VEL
LIN {X 0,Y 340.765,Z 734.04,A -85,B 0,C 180,E1 -14290.732,E2 -14290.732} C_VEL
LIN {X 0,Y 340.819,Z 734.031,A -85,B 0,C 180,E1 -14294.451,E2 -14294.451} C_VEL
LIN {X 0,Y 340.847,Z 734.025,A -85,B 0,C 180,E1 -14298.101,E2 -14298.101} C_VEL
LIN {X 0,Y 340.982,Z 734.008,A -85,B 0,C 180,E1 -14301.705,E2 -14301.705} C_VEL
LIN {X 0,Y 341.014,Z 734.004,A -85,B 0,C 180,E1 -14304.086,E2 -14304.086} C_VEL
LIN {X 0,Y 341.127,Z 733.991,A -85,B 0,C 180,E1 -14307.639,E2 -14307.639} C_VEL
LIN {X 0,Y 341.09,Z 733.999,A -85,B 0,C 180,E1 -14311.181,E2 -14311.181} C_VEL
LIN {X 0,Y 341.129,Z 733.989,A -85,B 0,C 180,E1 -14312.362,E2 -14312.362} C_VEL
LIN {X 0,Y 341.018,Z 734.004,A -85,B 0,C 180,E1 -14315.915,E2 -14315.915} C_VEL
LIN {X 0,Y 340.966,Z 734.009,A -85,B 0,C 180,E1 -14318.356,E2 -14318.356} C_VEL
LIN {X 0,Y 340.853,Z 734.026,A -85,B 0,C 180,E1 -14321.899,E2 -14321.899} C_VEL
LIN {X 0,Y 340.823,Z 734.033,A -85,B 0,C 180,E1 -14325.55,E2 -14325.55} C_VEL
LIN {X 0,Y 340.84,Z 734.025,A -85,B 0,C 180,E1 -14328.466,E2 -14328.466} C_VEL
LIN {X 0,Y 340.721,Z 734.046,A -85,B 0,C 180,E1 -14331.842,E2 -14331.842} C_VEL
LIN {X 0,Y 340.724,Z 734.044,A -85,B 0,C 180,E1 -14335.669,E2 -14335.669} C_VEL
LIN {X 0,Y 340.711,Z 734.044,A -85,B 0,C 180,E1 -14339.674,E2 -14339.674} C_VEL
LIN {X 0,Y 340.689,Z 734.046,A -85,B 0,C 180,E1 -14342.436,E2 -14342.436} C_VEL
LIN {X 0,Y 340.721,Z 734.04,A -85,B 0,C 180,E1 -14345.279,E2 -14345.279} C_VEL
LIN {X 0,Y 340.713,Z 734.045,A -85,B 0,C 180,E1 -14348.386,E2 -14348.386} C_VEL
LIN {X 0,Y 340.761,Z 734.038,A -85,B 0,C 180,E1 -14352.63,E2 -14352.63} C_VEL
LIN {X 0,Y 340.742,Z 734.04,A -85,B 0,C 180,E1 -14352.829,E2 -14352.829} C_VEL
LIN {X 0,Y 344.361,Z 746.61,A -85,B 0,C 180,E1 -14353.94,E2 -14353.94} C_VEL
LIN {X 0,Y 346.472,Z 754.427,A -85,B 0,C 180,E1 -14354.768,E2 -14354.768} C_VEL
LIN {X 0,Y 345.726,Z 765.186,A -85,B 0,C 180,E1 -14355.909,E2 -14355.909} C_VEL
LIN {X 0,Y 344.987,Z 774.871,A -85,B 0,C 180,E1 -14357.171,E2 -14357.171} C_VEL
LIN {X 0,Y 344.019,Z 785.198,A -85,B 0,C 180,E1 -14358.828,E2 -14358.828} C_VEL
LIN {X 0,Y 343.16,Z 794.057,A -85,B 0,C 180,E1 -14360.588,E2 -14360.588} C_VEL
LIN {X 0,Y 342.456,Z 801.226,A -85,B 0,C 180,E1 -14362.37,E2 -14362.37} C_VEL
LIN {X 0,Y 341.891,Z 806.952,A -85,B 0,C 180,E1 -14364.136,E2 -14364.136} C_VEL
LIN {X 0,Y 341.47,Z 812.236,A -85,B 0,C 180,E1 -14366.24,E2 -14366.24} C_VEL
LIN {X 0,Y 341.352,Z 813.811,A -85,B 0,C 180,E1 -14367.044,E2 -14367.044} C_VEL
LIN {X 0,Y 340.53,Z 815.559,A -85,B 0,C 180,E1 -14367.985,E2 -14367.985} C_VEL
LIN {X 0,Y 337.534,Z 818.043,A -85,B 0,C 180,E1 -14369.524,E2 -14369.524} C_VEL
LIN {X 0,Y 334.66,Z 819.863,A -85,B 0,C 180,E1 -14371.112,E2 -14371.112} C_VEL
LIN {X 0,Y 334.043,Z 820.431,A -85,B 0,C 180,E1 -14372.113,E2 -14372.113} C_VEL
LIN {X 0,Y 334.205,Z 820.699,A -85,B 0,C 180,E1 -14373.793,E2 -14373.793} C_VEL
LIN {X 0,Y 334.425,Z 820.306,A -85,B 0,C 180,E1 -14375.146,E2 -14375.146} C_VEL
LIN {X 0,Y 335.019,Z 818.596,A -85,B 0,C 180,E1 -14377.374,E2 -14377.374} C_VEL
LIN {X 0,Y 335.646,Z 816.186,A -85,B 0,C 180,E1 -14379.148,E2 -14379.148} C_VEL
LIN {X 0,Y 336.422,Z 812.421,A -85,B 0,C 180,E1 -14381.107,E2 -14381.107} C_VEL
LIN {X 0,Y 337.616,Z 806.705,A -85,B 0,C 180,E1 -14383.25,E2 -14383.25} C_VEL
LIN {X 0,Y 338.957,Z 799.58,A -85,B 0,C 180,E1 -14385.286,E2 -14385.286} C_VEL
LIN {X 0,Y 340.191,Z 792.572,A -85,B 0,C 180,E1 -14386.865,E2 -14386.865} C_VEL
LIN {X 0,Y 341.494,Z 784.065,A -85,B 0,C 180,E1 -14388.424,E2 -14388.424} C_VEL
LIN {X 0,Y 342.847,Z 774.065,A -85,B 0,C 180,E1 -14389.909,E2 -14389.909} C_VEL
LIN {X 0,Y 343.961,Z 763.803,A -85,B 0,C 180,E1 -14391.148,E2 -14391.148} C_VEL
LIN {X 0,Y 343.601,Z 761.252,A -85,B 0,C 180,E1 -14391.472,E2 -14391.472} C_VEL
LIN {X 0,Y 340.343,Z 750.418,A -85,B 0,C 180,E1 -14392.883,E2 -14392.883} C_VEL
LIN {X 0,Y 336.591,Z 741.093,A -85,B 0,C 180,E1 -14394.007,E2 -14394.007} C_VEL
LIN {X 0,Y 334.012,Z 735.653,A -85,B 0,C 180,E1 -14394.642,E2 -14394.642} C_VEL
LIN {X 0,Y 333.86,Z 734.895,A -85,B 0,C 180,E1 -14394.716,E2 -14394.716} C_VEL
LIN {X 0,Y 334.105,Z 734.869,A -85,B 0,C 180,E1 -14397.589,E2 -14397.589} C_VEL
LIN {X 0,Y 334.21,Z 734.856,A -85,B 0,C 180,E1 -14400,E2 -14400} C_VEL
LIN {X 0,Y 334.105,Z 734.862,A -85,B 0,C 180,E1 -14402.411,E2 -14402.411} C_VEL
LIN {X 0,Y 334.016,Z 734.872,A -85,B 0,C 180,E1 -14406.039,E2 -14406.039} C_VEL
LIN {X 0,Y 333.962,Z 734.878,A -85,B 0,C 180,E1 -14408.471,E2 -14408.471} C_VEL
LIN {X 0,Y 333.794,Z 734.9,A -85,B 0,C 180,E1 -14412.154,E2 -14412.154} C_VEL
LIN {X 0,Y 333.781,Z 734.903,A -85,B 0,C 180,E1 -14415.886,E2 -14415.886} C_VEL
LIN {X 0,Y 333.799,Z 734.901,A -85,B 0,C 180,E1 -14418.655,E2 -14418.655} C_VEL
LIN {X 0,Y 333.66,Z 734.924,A -85,B 0,C 180,E1 -14422.28,E2 -14422.28} C_VEL
LIN {X 0,Y 333.737,Z 734.909,A -85,B 0,C 180,E1 -14426.246,E2 -14426.246} C_VEL
LIN {X 0,Y 333.693,Z 734.915,A -85,B 0,C 180,E1 -14428.974,E2 -14428.974} C_VEL
LIN {X 0,Y 333.648,Z 734.924,A -85,B 0,C 180,E1 -14432.587,E2 -14432.587} C_VEL
LIN {X 0,Y 333.679,Z 734.926,A -85,B 0,C 180,E1 -14436.139,E2 -14436.139} C_VEL
LIN {X 0,Y 333.667,Z 735.104,A -85,B 0,C 180,E1 -14439.19,E2 -14439.19} C_VEL
LIN {X 0,Y 334.927,Z 740.587,A -85,B 0,C 180,E1 -14442.74,E2 -14442.74} C_VEL
LIN {X 0,Y 336.245,Z 747.17,A -85,B 0,C 180,E1 -14446.389,E2 -14446.389} C_VEL
LIN {X 0,Y 337.641,Z 754.183,A -85,B 0,C 180,E1 -14449.814,E2 -14449.814} C_VEL
LIN {X 0,Y 338.269,Z 759.458,A -85,B 0,C 180,E1 -14452.139,E2 -14452.139} C_VEL
LIN {X 0,Y 337.2,Z 766.879,A -85,B 0,C 180,E1 -14455.029,E2 -14455.029} C_VEL
LIN {X 0,Y 335.9,Z 776.168,A -85,B 0,C 180,E1 -14458.461,E2 -14458.461} C_VEL
LIN {X 0,Y 334.901,Z 786.533,A -85,B 0,C 180,E1 -14462.143,E2 -14462.143} C_VEL
LIN {X 0,Y 334.013,Z 797.145,A -85,B 0,C 180,E1 -14465.776,E2 -14465.776} C_VEL
LIN {X 0,Y 333.825,Z 800.305,A -85,B 0,C 180,E1 -14466.77,E2 -14466.77} C_VEL
LIN {X 0,Y 336.377,Z 814.35,A -85,B 0,C 180,E1 -14467.605,E2 -14467.605} C_VEL
LIN {X 0,Y 337.906,Z 828.047,A -85,B 0,C 180,E1 -14468.574,E2 -14468.574} C_VEL
LIN {X 0,Y 338.224,Z 841.628,A -85,B 0,C 180,E1 -14469.707,E2 -14469.707} C_VEL
LIN {X 0,Y 337.915,Z 853.273,A -85,B 0,C 180,E1 -14470.878,E2 -14470.878} C_VEL
LIN {X 0,Y 337.636,Z 862.278,A -85,B 0,C 180,E1 -14471.963,E2 -14471.963} C_VEL
LIN {X 0,Y 336.122,Z 871.993,A -85,B 0,C 180,E1 -14473.291,E2 -14473.291} C_VEL
LIN {X 0,Y 334.841,Z 881.661,A -85,B 0,C 180,E1 -14474.906,E2 -14474.906} C_VEL
LIN {X 0,Y 333.902,Z 890.015,A -85,B 0,C 180,E1 -14476.613,E2 -14476.613} C_VEL
LIN {X 0,Y 333.093,Z 898.459,A -85,B 0,C 180,E1 -14478.745,E2 -14478.745} C_VEL
LIN {X 0,Y 332.742,Z 905.106,A -85,B 0,C 180,E1 -14480.885,E2 -14480.885} C_VEL
LIN {X 0,Y 332.721,Z 910.317,A -85,B 0,C 180,E1 -14483.107,E2 -14483.107} C_VEL
LIN {X 0,Y 332.915,Z 913.787,A -85,B 0,C 180,E1 -14485.156,E2 -14485.156} C_VEL
LIN {X 0,Y 333.042,Z 915.272,A -85,B 0,C 180,E1 -14486.37,E2 -14486.37} C_VEL
LIN {X 0,Y 333.078,Z 916.276,A -85,B 0,C 180,E1 -14487.581,E2 -14487.581} C_VEL
LIN {X 0,Y 333.165,Z 916.859,A -85,B 0,C 180,E1 -14488.791,E2 -14488.791} C_VEL
LIN {X 0,Y 333.242,Z 917.027,A -85,B 0,C 180,E1 -14490,E2 -14490} C_VEL
LIN {X 0,Y 333.185,Z 916.757,A -85,B 0,C 180,E1 -14491.209,E2 -14491.209} C_VEL
LIN {X 0,Y 333.124,Z 916.016,A -85,B 0,C 180,E1 -14492.418,E2 -14492.418} C_VEL
LIN {X 0,Y 333.064,Z 914.84,A -85,B 0,C 180,E1 -14493.629,E2 -14493.629} C_VEL
LIN {X 0,Y 332.924,Z 912.224,A -85,B 0,C 180,E1 -14495.451,E2 -14495.451} C_VEL
LIN {X 0,Y 332.83,Z 908.52,A -85,B 0,C 180,E1 -14497.279,E2 -14497.279} C_VEL
LIN {X 0,Y 332.86,Z 903.644,A -85,B 0,C 180,E1 -14499.111,E2 -14499.111} C_VEL
LIN {X 0,Y 333.123,Z 897.471,A -85,B 0,C 180,E1 -14500.945,E2 -14500.945} C_VEL
LIN {X 0,Y 333.697,Z 889.797,A -85,B 0,C 180,E1 -14502.776,E2 -14502.776} C_VEL
LIN {X 0,Y 334.392,Z 881.95,A -85,B 0,C 180,E1 -14504.297,E2 -14504.297} C_VEL
LIN {X 0,Y 335.563,Z 871.386,A -85,B 0,C 180,E1 -14505.955,E2 -14505.955} C_VEL
LIN {X 0,Y 336.551,Z 861.98,A -85,B 0,C 180,E1 -14507.155,E2 -14507.155} C_VEL
LIN {X 0,Y 336.849,Z 854.973,A -85,B 0,C 180,E1 -14507.923,E2 -14507.923} C_VEL
LIN {X 0,Y 336.368,Z 842.767,A -85,B 0,C 180,E1 -14509.054,E2 -14509.054} C_VEL
LIN {X 0,Y 335.525,Z 829.149,A -85,B 0,C 180,E1 -14510.043,E2 -14510.043} C_VEL
LIN {X 0,Y 334.222,Z 815.094,A -85,B 0,C 180,E1 -14510.784,E2 -14510.784} C_VEL
LIN {X 0,Y 333.533,Z 807.992,A -85,B 0,C 180,E1 -14511.068,E2 -14511.068} C_VEL
LIN {X 0,Y 334.39,Z 795.433,A -85,B 0,C 180,E1 -14515.345,E2 -14515.345} C_VEL
LIN {X 0,Y 335.37,Z 785.344,A -85,B 0,C 180,E1 -14518.815,E2 -14518.815} C_VEL
LIN {X 0,Y 336.668,Z 773.737,A -85,B 0,C 180,E1 -14522.871,E2 -14522.871} C_VEL
LIN {X 0,Y 337.994,Z 763.987,A -85,B 0,C 180,E1 -14526.344,E2 -14526.344} C_VEL
LIN {X 0,Y 338.462,Z 759.697,A -85,B 0,C 180,E1 -14527.903,E2 -14527.903} C_VEL
LIN {X 0,Y 337.179,Z 752.397,A -85,B 0,C 180,E1 -14530.777,E2 -14530.777} C_VEL
LIN {X 0,Y 335.328,Z 743.269,A -85,B 0,C 180,E1 -14534.554,E2 -14534.554} C_VEL
LIN {X 0,Y 333.671,Z 734.923,A -85,B 0,C 180,E1 -14538.233,E2 -14538.233} C_VEL
LIN {X 0,Y 333.653,Z 734.921,A -85,B 0,C 180,E1 -14542.349,E2 -14542.349} C_VEL
LIN {X 0,Y 333.675,Z 734.92,A -85,B 0,C 180,E1 -14545.341,E2 -14545.341} C_VEL
LIN {X 0,Y 333.704,Z 734.919,A -85,B 0,C 180,E1 -14549.71,E2 -14549.71} C_VEL
LIN {X 0,Y 333.745,Z 734.91,A -85,B 0,C 180,E1 -14552.401,E2 -14552.401} C_VEL
LIN {X 0,Y 333.727,Z 734.911,A -85,B 0,C 180,E1 -14555.091,E2 -14555.091} C_VEL
LIN {X 0,Y 333.678,Z 734.917,A -85,B 0,C 180,E1 -14559.019,E2 -14559.019} C_VEL
LIN {X 0,Y 333.796,Z 734.904,A -85,B 0,C 180,E1 -14561.59,E2 -14561.59} C_VEL
LIN {X 0,Y 333.81,Z 734.901,A -85,B 0,C 180,E1 -14565.577,E2 -14565.577} C_VEL
LIN {X 0,Y 333.836,Z 734.898,A -85,B 0,C 180,E1 -14569.078,E2 -14569.078} C_VEL
LIN {X 0,Y 334.008,Z 734.88,A -85,B 0,C 180,E1 -14572.747,E2 -14572.747} C_VEL
LIN {X 0,Y 333.8,Z 734.903,A -85,B 0,C 180,E1 -14575.169,E2 -14575.169} C_VEL
LIN {X 0,Y 334.096,Z 734.865,A -85,B 0,C 180,E1 -14577.589,E2 -14577.589} C_VEL
LIN {X 0,Y 334.208,Z 734.852,A -85,B 0,C 180,E1 -14580,E2 -14580} C_VEL
LIN {X 0,Y 334.103,Z 734.867,A -85,B 0,C 180,E1 -14582.411,E2 -14582.411} C_VEL
LIN {X 0,Y 333.97,Z 734.88,A -85,B 0,C 180,E1 -14586.52,E2 -14586.52} C_VEL
LIN {X 0,Y 333.822,Z 734.9,A -85,B 0,C 180,E1 -14589.696,E2 -14589.696} C_VEL
LIN {X 0,Y 333.799,Z 734.905,A -85,B 0,C 180,E1 -14593.392,E2 -14593.392} C_VEL
LIN {X 0,Y 333.722,Z 734.918,A -85,B 0,C 180,E1 -14597.148,E2 -14597.148} C_VEL
LIN {X 0,Y 333.691,Z 734.917,A -85,B 0,C 180,E1 -14599.693,E2 -14599.693} C_VEL
LIN {X 0,Y 333.644,Z 734.925,A -85,B 0,C 180,E1 -14603.592,E2 -14603.592} C_VEL
LIN {X 0,Y 333.67,Z 734.923,A -85,B 0,C 180,E1 -14607.606,E2 -14607.606} C_VEL
LIN {X 0,Y 333.659,Z 734.92,A -85,B 0,C 180,E1 -14610.366,E2 -14610.366} C_VEL
LIN {X 0,Y 333.638,Z 734.925,A -85,B 0,C 180,E1 -14613.209,E2 -14613.209} C_VEL
LIN {X 0,Y 333.675,Z 734.919,A -85,B 0,C 180,E1 -14616.14,E2 -14616.14} C_VEL
LIN {X 0,Y 333.603,Z 734.928,A -85,B 0,C 180,E1 -14619.199,E2 -14619.199} C_VEL
LIN {X 0,Y 333.628,Z 734.924,A -85,B 0,C 180,E1 -14622.499,E2 -14622.499} C_VEL
LIN {X 0,Y 333.595,Z 734.933,A -85,B 0,C 180,E1 -14625.955,E2 -14625.955} C_VEL
LIN {X 0,Y 333.603,Z 734.927,A -85,B 0,C 180,E1 -14629.325,E2 -14629.325} C_VEL
LIN {X 0,Y 333.663,Z 734.919,A -85,B 0,C 180,E1 -14633.169,E2 -14633.169} C_VEL
LIN {X 0,Y 333.674,Z 734.918,A -85,B 0,C 180,E1 -14635.341,E2 -14635.341} C_VEL
LIN {X 0,Y 333.631,Z 734.929,A -85,B 0,C 180,E1 -14638.222,E2 -14638.222} C_VEL
LIN {X 0,Y 333.631,Z 734.924,A -85,B 0,C 180,E1 -14641.02,E2 -14641.02} C_VEL
LIN {X 0,Y 333.659,Z 734.922,A -85,B 0,C 180,E1 -14644.922,E2 -14644.922} C_VEL
LIN {X 0,Y 333.668,Z 734.92,A -85,B 0,C 180,E1 -14649.018,E2 -14649.018} C_VEL
LIN {X 0,Y 333.744,Z 734.909,A -85,B 0,C 180,E1 -14651.587,E2 -14651.587} C_VEL
LIN {X 0,Y 333.811,Z 734.901,A -85,B 0,C 180,E1 -14655.577,E2 -14655.577} C_VEL
LIN {X 0,Y 333.816,Z 734.904,A -85,B 0,C 180,E1 -14659.078,E2 -14659.078} C_VEL
LIN {X 0,Y 333.958,Z 734.886,A -85,B 0,C 180,E1 -14662.746,E2 -14662.746} C_VEL
LIN {X 0,Y 333.778,Z 734.91,A -85,B 0,C 180,E1 -14665.169,E2 -14665.169} C_VEL
LIN {X 0,Y 334.067,Z 734.87,A -85,B 0,C 180,E1 -14667.589,E2 -14667.589} C_VEL
LIN {X 0,Y 334.061,Z 734.875,A -85,B 0,C 180,E1 -14671.206,E2 -14671.206} C_VEL
LIN {X 0,Y 334.069,Z 734.869,A -85,B 0,C 180,E1 -14672.412,E2 -14672.412} C_VEL
LIN {X 0,Y 333.992,Z 734.879,A -85,B 0,C 180,E1 -14676.04,E2 -14676.04} C_VEL
LIN {X 0,Y 333.823,Z 734.903,A -85,B 0,C 180,E1 -14679.696,E2 -14679.696} C_VEL
LIN {X 0,Y 333.8,Z 734.907,A -85,B 0,C 180,E1 -14683.391,E2 -14683.391} C_VEL
LIN {X 0,Y 333.75,Z 734.91,A -85,B 0,C 180,E1 -14687.146,E2 -14687.146} C_VEL
LIN {X 0,Y 333.735,Z 734.916,A -85,B 0,C 180,E1 -14689.691,E2 -14689.691} C_VEL
LIN {X 0,Y 333.66,Z 734.923,A -85,B 0,C 180,E1 -14693.591,E2 -14693.591} C_VEL
LIN {X 0,Y 333.66,Z 734.922,A -85,B 0,C 180,E1 -14696.253,E2 -14696.253} C_VEL
LIN {X 0,Y 333.665,Z 734.922,A -85,B 0,C 180,E1 -14700.278,E2 -14700.278} C_VEL
LIN {X 0,Y 333.64,Z 734.922,A -85,B 0,C 180,E1 -14703.208,E2 -14703.208} C_VEL
LIN {X 0,Y 333.679,Z 734.923,A -85,B 0,C 180,E1 -14706.139,E2 -14706.139} C_VEL
LIN {X 0,Y 333.65,Z 734.92,A -85,B 0,C 180,E1 -14709.192,E2 -14709.192} C_VEL
LIN {X 0,Y 333.721,Z 734.916,A -85,B 0,C 180,E1 -14712.491,E2 -14712.491} C_VEL
LIN {X 0,Y 337.361,Z 747.471,A -85,B 0,C 180,E1 -14713.635,E2 -14713.635} C_VEL
LIN {X 0,Y 339.539,Z 755.639,A -85,B 0,C 180,E1 -14714.521,E2 -14714.521} C_VEL
LIN {X 0,Y 338.878,Z 765.769,A -85,B 0,C 180,E1 -14715.619,E2 -14715.619} C_VEL
LIN {X 0,Y 338.001,Z 776.704,A -85,B 0,C 180,E1 -14717.08,E2 -14717.08} C_VEL
LIN {X 0,Y 337.083,Z 786.192,A -85,B 0,C 180,E1 -14718.641,E2 -14718.641} C_VEL
LIN {X 0,Y 336.253,Z 794.413,A -85,B 0,C 180,E1 -14720.291,E2 -14720.291} C_VEL
LIN {X 0,Y 335.474,Z 802.085,A -85,B 0,C 180,E1 -14722.209,E2 -14722.209} C_VEL
LIN {X 0,Y 334.897,Z 807.847,A -85,B 0,C 180,E1 -14724.013,E2 -14724.013} C_VEL
LIN {X 0,Y 334.448,Z 813.17,A -85,B 0,C 180,E1 -14726.16,E2 -14726.16} C_VEL
LIN {X 0,Y 334.135,Z 816.927,A -85,B 0,C 180,E1 -14728.275,E2 -14728.275} C_VEL
LIN {X 0,Y 334.003,Z 818.675,A -85,B 0,C 180,E1 -14729.668,E2 -14729.668} C_VEL
LIN {X 0,Y 333.976,Z 819.886,A -85,B 0,C 180,E1 -14731.053,E2 -14731.053} C_VEL
LIN {X 0,Y 334.043,Z 820.431,A -85,B 0,C 180,E1 -14732.113,E2 -14732.113} C_VEL
LIN {X 0,Y 333.481,Z 820.778,A -85,B 0,C 180,E1 -14733.122,E2 -14733.122} C_VEL
LIN {X 0,Y 330.908,Z 821.1,A -85,B 0,C 180,E1 -14734.773,E2 -14734.773} C_VEL
LIN {X 0,Y 328.443,Z 820.675,A -85,B 0,C 180,E1 -14736.441,E2 -14736.441} C_VEL
LIN {X 0,Y 328.056,Z 819.801,A -85,B 0,C 180,E1 -14737.459,E2 -14737.459} C_VEL
LIN {X 0,Y 328.746,Z 817.392,A -85,B 0,C 180,E1 -14739.345,E2 -14739.345} C_VEL
LIN {X 0,Y 329.582,Z 813.677,A -85,B 0,C 180,E1 -14741.345,E2 -14741.345} C_VEL
LIN {X 0,Y 330.836,Z 808.015,A -85,B 0,C 180,E1 -14743.533,E2 -14743.533} C_VEL
LIN {X 0,Y 332.24,Z 800.998,A -85,B 0,C 180,E1 -14745.592,E2 -14745.592} C_VEL
LIN {X 0,Y 333.556,Z 793.98,A -85,B 0,C 180,E1 -14747.218,E2 -14747.218} C_VEL
LIN {X 0,Y 334.936,Z 785.58,A -85,B 0,C 180,E1 -14748.808,E2 -14748.808} C_VEL
LIN {X 0,Y 336.226,Z 776.745,A -85,B 0,C 180,E1 -14750.176,E2 -14750.176} C_VEL
LIN {X 0,Y 337.625,Z 765.201,A -85,B 0,C 180,E1 -14751.621,E2 -14751.621} C_VEL
LIN {X 0,Y 334.967,Z 755.721,A -85,B 0,C 180,E1 -14752.938,E2 -14752.938} C_VEL
LIN {X 0,Y 331.436,Z 746.12,A -85,B 0,C 180,E1 -14754.188,E2 -14754.188} C_VEL
LIN {X 0,Y 328.076,Z 739.094,A -85,B 0,C 180,E1 -14755.084,E2 -14755.084} C_VEL
LIN {X 0,Y 326.812,Z 736.178,A -85,B 0,C 180,E1 -14755.413,E2 -14755.413} C_VEL
LIN {X 0,Y 326.773,Z 735.783,A -85,B 0,C 180,E1 -14755.451,E2 -14755.451} C_VEL
LIN {X 0,Y 327.045,Z 735.748,A -85,B 0,C 180,E1 -14757.537,E2 -14757.537} C_VEL
LIN {X 0,Y 327.162,Z 735.734,A -85,B 0,C 180,E1 -14760,E2 -14760} C_VEL
LIN {X 0,Y 327.046,Z 735.741,A -85,B 0,C 180,E1 -14762.463,E2 -14762.463} C_VEL
LIN {X 0,Y 326.99,Z 735.747,A -85,B 0,C 180,E1 -14766.169,E2 -14766.169} C_VEL
LIN {X 0,Y 326.809,Z 735.772,A -85,B 0,C 180,E1 -14769.906,E2 -14769.906} C_VEL
LIN {X 0,Y 326.762,Z 735.783,A -85,B 0,C 180,E1 -14773.685,E2 -14773.685} C_VEL
LIN {X 0,Y 326.702,Z 735.786,A -85,B 0,C 180,E1 -14777.528,E2 -14777.528} C_VEL
LIN {X 0,Y 326.661,Z 735.793,A -85,B 0,C 180,E1 -14780.135,E2 -14780.135} C_VEL
LIN {X 0,Y 326.652,Z 735.791,A -85,B 0,C 180,E1 -14784.129,E2 -14784.129} C_VEL
LIN {X 0,Y 326.685,Z 735.788,A -85,B 0,C 180,E1 -14786.858,E2 -14786.858} C_VEL
LIN {X 0,Y 326.636,Z 735.796,A -85,B 0,C 180,E1 -14790.61,E2 -14790.61} C_VEL
LIN {X 0,Y 326.61,Z 735.803,A -85,B 0,C 180,E1 -14794.019,E2 -14794.019} C_VEL
LIN {X 0,Y 326.595,Z 735.81,A -85,B 0,C 180,E1 -14798.054,E2 -14798.054} C_VEL
LIN {X 0,Y 327.745,Z 740.976,A -85,B 0,C 180,E1 -14801.663,E2 -14801.663} C_VEL
LIN {X 0,Y 328.985,Z 746.88,A -85,B 0,C 180,E1 -14805.173,E2 -14805.173} C_VEL
LIN {X 0,Y 330.326,Z 753.744,A -85,B 0,C 180,E1 -14808.734,E2 -14808.734} C_VEL
LIN {X 0,Y 331.239,Z 758.897,A -85,B 0,C 180,E1 -14811.16,E2 -14811.16} C_VEL
LIN {X 0,Y 331.33,Z 760.889,A -85,B 0,C 180,E1 -14812.038,E2 -14812.038} C_VEL
LIN {X 0,Y 330.246,Z 768.133,A -85,B 0,C 180,E1 -14814.929,E2 -14814.929} C_VEL
LIN {X 0,Y 328.703,Z 779.245,A -85,B 0,C 180,E1 -14819.126,E2 -14819.126} C_VEL
LIN {X 0,Y 327.546,Z 790.61,A -85,B 0,C 180,E1 -14823.218,E2 -14823.218} C_VEL
LIN {X 0,Y 326.873,Z 798.702,A -85,B 0,C 180,E1 -14826.04,E2 -14826.04} C_VEL
LIN {X 0,Y 329.64,Z 813.751,A -85,B 0,C 180,E1 -14826.998,E2 -14826.998} C_VEL
LIN {X 0,Y 331.202,Z 827.173,A -85,B 0,C 180,E1 -14827.992,E2 -14827.992} C_VEL
LIN {X 0,Y 331.542,Z 839.172,A -85,B 0,C 180,E1 -14829.024,E2 -14829.024} C_VEL
LIN {X 0,Y 331.131,Z 851.709,A -85,B 0,C 180,E1 -14830.31,E2 -14830.31} C_VEL
LIN {X 0,Y 330.705,Z 863.128,A -85,B 0,C 180,E1 -14831.732,E2 -14831.732} C_VEL
LIN {X 0,Y 329.016,Z 873.435,A -85,B 0,C 180,E1 -14833.239,E2 -14833.239} C_VEL
LIN {X 0,Y 327.513,Z 883.587,A -85,B 0,C 180,E1 -14835.078,E2 -14835.078} C_VEL
LIN {X 0,Y 326.762,Z 890.611,A -85,B 0,C 180,E1 -14836.631,E2 -14836.631} C_VEL
LIN {X 0,Y 326.093,Z 897.652,A -85,B 0,C 180,E1 -14838.5,E2 -14838.5} C_VEL
LIN {X 0,Y 325.674,Z 904.21,A -85,B 0,C 180,E1 -14840.686,E2 -14840.686} C_VEL
LIN {X 0,Y 325.611,Z 908.6,A -85,B 0,C 180,E1 -14842.559,E2 -14842.559} C_VEL
LIN {X 0,Y 325.704,Z 910.926,A -85,B 0,C 180,E1 -14843.806,E2 -14843.806} C_VEL
LIN {X 0,Y 325.843,Z 912.825,A -85,B 0,C 180,E1 -14845.051,E2 -14845.051} C_VEL
LIN {X 0,Y 325.998,Z 914.283,A -85,B 0,C 180,E1 -14846.292,E2 -14846.292} C_VEL
LIN {X 0,Y 326.038,Z 915.257,A -85,B 0,C 180,E1 -14847.529,E2 -14847.529} C_VEL
LIN {X 0,Y 326.132,Z 915.824,A -85,B 0,C 180,E1 -14848.765,E2 -14848.765} C_VEL
LIN {X 0,Y 326.244,Z 915.981,A -85,B 0,C 180,E1 -14850,E2 -14850} C_VEL
LIN {X 0,Y 326.159,Z 915.679,A -85,B 0,C 180,E1 -14851.235,E2 -14851.235} C_VEL
LIN {X 0,Y 326.091,Z 914.91,A -85,B 0,C 180,E1 -14852.47,E2 -14852.47} C_VEL
LIN {X 0,Y 326.022,Z 913.715,A -85,B 0,C 180,E1 -14853.708,E2 -14853.708} C_VEL
LIN {X 0,Y 325.878,Z 911.057,A -85,B 0,C 180,E1 -14855.569,E2 -14855.569} C_VEL
LIN {X 0,Y 325.794,Z 907.306,A -85,B 0,C 180,E1 -14857.437,E2 -14857.437} C_VEL
LIN {X 0,Y 325.795,Z 902.368,A -85,B 0,C 180,E1 -14859.311,E2 -14859.311} C_VEL
LIN {X 0,Y 326.083,Z 896.133,A -85,B 0,C 180,E1 -14861.185,E2 -14861.185} C_VEL
LIN {X 0,Y 326.723,Z 888.363,A -85,B 0,C 180,E1 -14863.053,E2 -14863.053} C_VEL
LIN {X 0,Y 327.426,Z 880.416,A -85,B 0,C 180,E1 -14864.608,E2 -14864.608} C_VEL
LIN {X 0,Y 328.531,Z 870.815,A -85,B 0,C 180,E1 -14866.147,E2 -14866.147} C_VEL
LIN {X 0,Y 329.762,Z 860.252,A -85,B 0,C 180,E1 -14867.52,E2 -14867.52} C_VEL
LIN {X 0,Y 329.63,Z 851.355,A -85,B 0,C 180,E1 -14868.49,E2 -14868.49} C_VEL
LIN {X 0,Y 329.183,Z 839.777,A -85,B 0,C 180,E1 -14869.543,E2 -14869.543} C_VEL
LIN {X 0,Y 328.393,Z 827.288,A -85,B 0,C 180,E1 -14870.433,E2 -14870.433} C_VEL
LIN {X 0,Y 327.06,Z 812.829,A -85,B 0,C 180,E1 -14871.199,E2 -14871.199} C_VEL
LIN {X 0,Y 326.486,Z 807.01,A -85,B 0,C 180,E1 -14871.466,E2 -14871.466} C_VEL
LIN {X 0,Y 327.394,Z 795.063,A -85,B 0,C 180,E1 -14875.632,E2 -14875.632} C_VEL
LIN {X 0,Y 328.477,Z 784.174,A -85,B 0,C 180,E1 -14879.479,E2 -14879.479} C_VEL
LIN {X 0,Y 329.947,Z 772.055,A -85,B 0,C 180,E1 -14883.827,E2 -14883.827} C_VEL
LIN {X 0,Y 331.281,Z 762.841,A -85,B 0,C 180,E1 -14887.201,E2 -14887.201} C_VEL
LIN {X 0,Y 331.35,Z 759.943,A -85,B 0,C 180,E1 -14888.3,E2 -14888.3} C_VEL
LIN {X 0,Y 329.748,Z 751.415,A -85,B 0,C 180,E1 -14891.758,E2 -14891.758} C_VEL
LIN {X 0,Y 327.813,Z 741.944,A -85,B 0,C 180,E1 -14895.832,E2 -14895.832} C_VEL
LIN {X 0,Y 326.612,Z 735.802,A -85,B 0,C 180,E1 -14898.665,E2 -14898.665} C_VEL
LIN {X 0,Y 326.625,Z 735.8,A -85,B 0,C 180,E1 -14901.392,E2 -14901.392} C_VEL
LIN {X 0,Y 326.62,Z 735.796,A -85,B 0,C 180,E1 -14904.851,E2 -14904.851} C_VEL
LIN {X 0,Y 326.611,Z 735.8,A -85,B 0,C 180,E1 -14907.456,E2 -14907.456} C_VEL
LIN {X 0,Y 326.662,Z 735.793,A -85,B 0,C 180,E1 -14910.341,E2 -14910.341} C_VEL
LIN {X 0,Y 326.691,Z 735.789,A -85,B 0,C 180,E1 -14914.516,E2 -14914.516} C_VEL
LIN {X 0,Y 326.623,Z 735.798,A -85,B 0,C 180,E1 -14918.544,E2 -14918.544} C_VEL
LIN {X 0,Y 326.746,Z 735.78,A -85,B 0,C 180,E1 -14921.178,E2 -14921.178} C_VEL
LIN {X 0,Y 326.765,Z 735.778,A -85,B 0,C 180,E1 -14925.433,E2 -14925.433} C_VEL
LIN {X 0,Y 326.772,Z 735.779,A -85,B 0,C 180,E1 -14928.839,E2 -14928.839} C_VEL
LIN {X 0,Y 326.96,Z 735.759,A -85,B 0,C 180,E1 -14932.59,E2 -14932.59} C_VEL
LIN {X 0,Y 326.99,Z 735.751,A -85,B 0,C 180,E1 -14933.831,E2 -14933.831} C_VEL
LIN {X 0,Y 327.036,Z 735.744,A -85,B 0,C 180,E1 -14937.537,E2 -14937.537} C_VEL
LIN {X 0,Y 327.161,Z 735.729,A -85,B 0,C 180,E1 -14940,E2 -14940} C_VEL
LIN {X 0,Y 327.044,Z 735.747,A -85,B 0,C 180,E1 -14942.463,E2 -14942.463} C_VEL
LIN {X 0,Y 326.93,Z 735.756,A -85,B 0,C 180,E1 -14946.509,E2 -14946.509} C_VEL
LIN {X 0,Y 326.785,Z 735.776,A -85,B 0,C 180,E1 -14949.907,E2 -14949.907} C_VEL
LIN {X 0,Y 326.761,Z 735.779,A -85,B 0,C 180,E1 -14953.685,E2 -14953.685} C_VEL
LIN {X 0,Y 326.666,Z 735.793,A -85,B 0,C 180,E1 -14957.53,E2 -14957.53} C_VEL
LIN {X 0,Y 326.633,Z 735.795,A -85,B 0,C 180,E1 -14960.137,E2 -14960.137} C_VEL
LIN {X 0,Y 326.592,Z 735.801,A -85,B 0,C 180,E1 -14962.79,E2 -14962.79} C_VEL
LIN {X 0,Y 326.603,Z 735.803,A -85,B 0,C 180,E1 -14965.491,E2 -14965.491} C_VEL
LIN {X 0,Y 326.619,Z 735.801,A -85,B 0,C 180,E1 -14969.664,E2 -14969.664} C_VEL
LIN {X 0,Y 326.619,Z 735.797,A -85,B 0,C 180,E1 -14972.946,E2 -14972.946} C_VEL
LIN {X 0,Y 326.612,Z 735.802,A -85,B 0,C 180,E1 -14975.52,E2 -14975.52} C_VEL
LIN {X 0,Y 326.572,Z 735.803,A -85,B 0,C 180,E1 -14979.219,E2 -14979.219} C_VEL
LIN {X 0,Y 326.573,Z 735.802,A -85,B 0,C 180,E1 -14982.971,E2 -14982.971} C_VEL
LIN {X 0,Y 326.573,Z 735.802,A -85,B 0,C 180,E1 -14987.029,E2 -14987.029} C_VEL
LIN {X 0,Y 326.572,Z 735.803,A -85,B 0,C 180,E1 -14990.782,E2 -14990.782} C_VEL
LIN {X 0,Y 326.612,Z 735.8,A -85,B 0,C 180,E1 -14994.48,E2 -14994.48} C_VEL
LIN {X 0,Y 326.609,Z 735.798,A -85,B 0,C 180,E1 -14997.456,E2 -14997.456} C_VEL
LIN {X 0,Y 326.582,Z 735.807,A -85,B 0,C 180,E1 -15000.333,E2 -15000.333} C_VEL
LIN {X 0,Y 326.598,Z 735.799,A -85,B 0,C 180,E1 -15003.135,E2 -15003.135} C_VEL
LIN {X 0,Y 326.593,Z 735.8,A -85,B 0,C 180,E1 -15007.211,E2 -15007.211} C_VEL
LIN {X 0,Y 326.709,Z 735.786,A -85,B 0,C 180,E1 -15011.175,E2 -15011.175} C_VEL
LIN {X 0,Y 326.766,Z 735.779,A -85,B 0,C 180,E1 -15015.433,E2 -15015.433} C_VEL
LIN {X 0,Y 326.757,Z 735.785,A -85,B 0,C 180,E1 -15018.839,E2 -15018.839} C_VEL
LIN {X 0,Y 326.915,Z 735.762,A -85,B 0,C 180,E1 -15022.589,E2 -15022.589} C_VEL
LIN {X 0,Y 326.747,Z 735.786,A -85,B 0,C 180,E1 -15025.065,E2 -15025.065} C_VEL
LIN {X 0,Y 327.01,Z 735.75,A -85,B 0,C 180,E1 -15027.537,E2 -15027.537} C_VEL
LIN {X 0,Y 327.031,Z 735.751,A -85,B 0,C 180,E1 -15031.232,E2 -15031.232} C_VEL
LIN {X 0,Y 326.756,Z 735.781,A -85,B 0,C 180,E1 -15033.7,E2 -15033.7} C_VEL
LIN {X 0,Y 326.946,Z 735.756,A -85,B 0,C 180,E1 -15036.17,E2 -15036.17} C_VEL
LIN {X 0,Y 326.786,Z 735.777,A -85,B 0,C 180,E1 -15039.907,E2 -15039.907} C_VEL
LIN {X 0,Y 326.762,Z 735.783,A -85,B 0,C 180,E1 -15043.685,E2 -15043.685} C_VEL
LIN {X 0,Y 326.703,Z 735.791,A -85,B 0,C 180,E1 -15047.528,E2 -15047.528} C_VEL
LIN {X 0,Y 326.659,Z 735.794,A -85,B 0,C 180,E1 -15050.135,E2 -15050.135} C_VEL
LIN {X 0,Y 326.634,Z 735.798,A -85,B 0,C 180,E1 -15054.131,E2 -15054.131} C_VEL
LIN {X 0,Y 326.606,Z 735.803,A -85,B 0,C 180,E1 -15058.084,E2 -15058.084} C_VEL
LIN {X 0,Y 326.576,Z 735.802,A -85,B 0,C 180,E1 -15061.097,E2 -15061.097} C_VEL
LIN {X 0,Y 326.61,Z 735.803,A -85,B 0,C 180,E1 -15064.019,E2 -15064.019} C_VEL
LIN {X 0,Y 326.63,Z 735.795,A -85,B 0,C 180,E1 -15067.239,E2 -15067.239} C_VEL
LIN {X 0,Y 326.593,Z 735.8,A -85,B 0,C 180,E1 -15071.134,E2 -15071.134} C_VEL
LIN {X 0,Y 326.632,Z 735.804,A -85,B 0,C 180,E1 -15072.174,E2 -15072.174} C_VEL
LIN {X 0,Y 330.377,Z 748.629,A -85,B 0,C 180,E1 -15073.36,E2 -15073.36} C_VEL
LIN {X 0,Y 332.523,Z 756.431,A -85,B 0,C 180,E1 -15074.225,E2 -15074.225} C_VEL
LIN {X 0,Y 332.529,Z 760.197,A -85,B 0,C 180,E1 -15074.628,E2 -15074.628} C_VEL
LIN {X 0,Y 331.592,Z 771.239,A -85,B 0,C 180,E1 -15075.944,E2 -15075.944} C_VEL
LIN {X 0,Y 330.727,Z 781.566,A -85,B 0,C 180,E1 -15077.477,E2 -15077.477} C_VEL
LIN {X 0,Y 329.813,Z 790.301,A -85,B 0,C 180,E1 -15079.061,E2 -15079.061} C_VEL
LIN {X 0,Y 328.944,Z 798.71,A -85,B 0,C 180,E1 -15080.929,E2 -15080.929} C_VEL
LIN {X 0,Y 328.278,Z 805.317,A -85,B 0,C 180,E1 -15082.758,E2 -15082.758} C_VEL
LIN {X 0,Y 327.721,Z 810.687,A -85,B 0,C 180,E1 -15084.618,E2 -15084.618} C_VEL
LIN {X 0,Y 327.327,Z 815.616,A -85,B 0,C 180,E1 -15086.864,E2 -15086.864} C_VEL
LIN {X 0,Y 327.036,Z 818.877,A -85,B 0,C 180,E1 -15088.951,E2 -15088.951} C_VEL
LIN {X 0,Y 326.945,Z 820.361,A -85,B 0,C 180,E1 -15090.369,E2 -15090.369} C_VEL
LIN {X 0,Y 327.021,Z 821.43,A -85,B 0,C 180,E1 -15092.113,E2 -15092.113} C_VEL
LIN {X 0,Y 327.123,Z 821.75,A -85,B 0,C 180,E1 -15093.181,E2 -15093.181} C_VEL
LIN {X 0,Y 327.331,Z 821.66,A -85,B 0,C 180,E1 -15094.569,E2 -15094.569} C_VEL
LIN {X 0,Y 327.612,Z 821.082,A -85,B 0,C 180,E1 -15095.946,E2 -15095.946} C_VEL
LIN {X 0,Y 328.056,Z 819.801,A -85,B 0,C 180,E1 -15097.459,E2 -15097.459} C_VEL
LIN {X 0,Y 327.72,Z 818.801,A -85,B 0,C 180,E1 -15098.471,E2 -15098.471} C_VEL
LIN {X 0,Y 325.557,Z 816.88,A -85,B 0,C 180,E1 -15100.135,E2 -15100.135} C_VEL
LIN {X 0,Y 323.805,Z 814.923,A -85,B 0,C 180,E1 -15101.458,E2 -15101.458} C_VEL
LIN {X 0,Y 323.303,Z 812.977,A -85,B 0,C 180,E1 -15102.444,E2 -15102.444} C_VEL
LIN {X 0,Y 323.4,Z 812.19,A -85,B 0,C 180,E1 -15102.767,E2 -15102.767} C_VEL
LIN {X 0,Y 324.61,Z 806.929,A -85,B 0,C 180,E1 -15104.62,E2 -15104.62} C_VEL
LIN {X 0,Y 326.131,Z 799.716,A -85,B 0,C 180,E1 -15106.605,E2 -15106.605} C_VEL
LIN {X 0,Y 327.482,Z 792.357,A -85,B 0,C 180,E1 -15108.236,E2 -15108.236} C_VEL
LIN {X 0,Y 329.027,Z 783.34,A -85,B 0,C 180,E1 -15109.85,E2 -15109.85} C_VEL
LIN {X 0,Y 330.467,Z 773.395,A -85,B 0,C 180,E1 -15111.284,E2 -15111.284} C_VEL
LIN {X 0,Y 331.167,Z 767.801,A -85,B 0,C 180,E1 -15111.972,E2 -15111.972} C_VEL
LIN {X 0,Y 328.98,Z 759.062,A -85,B 0,C 180,E1 -15113.252,E2 -15113.252} C_VEL
LIN {X 0,Y 325.368,Z 749.07,A -85,B 0,C 180,E1 -15114.638,E2 -15114.638} C_VEL
LIN {X 0,Y 319.985,Z 737.772,A -85,B 0,C 180,E1 -15116.143,E2 -15116.143} C_VEL
LIN {X 0,Y 319.74,Z 736.658,A -85,B 0,C 180,E1 -15116.298,E2 -15116.298} C_VEL
LIN {X 0,Y 320.02,Z 736.623,A -85,B 0,C 180,E1 -15118.741,E2 -15118.741} C_VEL
LIN {X 0,Y 320.022,Z 736.621,A -85,B 0,C 180,E1 -15121.258,E2 -15121.258} C_VEL
LIN {X 0,Y 319.738,Z 736.653,A -85,B 0,C 180,E1 -15123.781,E2 -15123.781} C_VEL
LIN {X 0,Y 319.945,Z 736.625,A -85,B 0,C 180,E1 -15126.305,E2 -15126.305} C_VEL
LIN {X 0,Y 319.84,Z 736.635,A -85,B 0,C 180,E1 -15128.848,E2 -15128.848} C_VEL
LIN {X 0,Y 319.685,Z 736.659,A -85,B 0,C 180,E1 -15132.7,E2 -15132.7} C_VEL
LIN {X 0,Y 319.703,Z 736.653,A -85,B 0,C 180,E1 -15135.295,E2 -15135.295} C_VEL
LIN {X 0,Y 319.676,Z 736.664,A -85,B 0,C 180,E1 -15139.255,E2 -15139.255} C_VEL
LIN {X 0,Y 319.563,Z 736.675,A -85,B 0,C 180,E1 -15143.32,E2 -15143.32} C_VEL
LIN {X 0,Y 319.621,Z 736.668,A -85,B 0,C 180,E1 -15146.089,E2 -15146.089} C_VEL
LIN {X 0,Y 319.582,Z 736.672,A -85,B 0,C 180,E1 -15148.934,E2 -15148.934} C_VEL
LIN {X 0,Y 319.534,Z 736.682,A -85,B 0,C 180,E1 -15151.862,E2 -15151.862} C_VEL
LIN {X 0,Y 319.582,Z 736.677,A -85,B 0,C 180,E1 -15155.543,E2 -15155.543} C_VEL
LIN {X 0,Y 319.601,Z 736.745,A -85,B 0,C 180,E1 -15157.065,E2 -15157.065} C_VEL
LIN {X 0,Y 320.784,Z 742.229,A -85,B 0,C 180,E1 -15161.092,E2 -15161.092} C_VEL
LIN {X 0,Y 321.894,Z 747.404,A -85,B 0,C 180,E1 -15164.32,E2 -15164.32} C_VEL
LIN {X 0,Y 323.076,Z 753.545,A -85,B 0,C 180,E1 -15167.699,E2 -15167.699} C_VEL
LIN {X 0,Y 324.065,Z 758.681,A -85,B 0,C 180,E1 -15170.261,E2 -15170.261} C_VEL
LIN {X 0,Y 324.407,Z 762.433,A -85,B 0,C 180,E1 -15171.966,E2 -15171.966} C_VEL
LIN {X 0,Y 323.287,Z 769.405,A -85,B 0,C 180,E1 -15174.824,E2 -15174.824} C_VEL
LIN {X 0,Y 321.672,Z 780.458,A -85,B 0,C 180,E1 -15179.107,E2 -15179.107} C_VEL
LIN {X 0,Y 320.655,Z 789.875,A -85,B 0,C 180,E1 -15182.595,E2 -15182.595} C_VEL
LIN {X 0,Y 319.98,Z 797.273,A -85,B 0,C 180,E1 -15185.258,E2 -15185.258} C_VEL
LIN {X 0,Y 323.03,Z 813.14,A -85,B 0,C 180,E1 -15186.35,E2 -15186.35} C_VEL
LIN {X 0,Y 324.454,Z 825.55,A -85,B 0,C 180,E1 -15187.323,E2 -15187.323} C_VEL
LIN {X 0,Y 324.89,Z 837.945,A -85,B 0,C 180,E1 -15188.423,E2 -15188.423} C_VEL
LIN {X 0,Y 324.465,Z 850.337,A -85,B 0,C 180,E1 -15189.722,E2 -15189.722} C_VEL
LIN {X 0,Y 324.056,Z 861.706,A -85,B 0,C 180,E1 -15191.179,E2 -15191.179} C_VEL
LIN {X 0,Y 322.509,Z 871.09,A -85,B 0,C 180,E1 -15192.564,E2 -15192.564} C_VEL
LIN {X 0,Y 321.006,Z 880.918,A -85,B 0,C 180,E1 -15194.337,E2 -15194.337} C_VEL
LIN {X 0,Y 320.217,Z 887.334,A -85,B 0,C 180,E1 -15195.713,E2 -15195.713} C_VEL
LIN {X 0,Y 319.312,Z 894.706,A -85,B 0,C 180,E1 -15197.608,E2 -15197.608} C_VEL
LIN {X 0,Y 318.698,Z 901.661,A -85,B 0,C 180,E1 -15199.839,E2 -15199.839} C_VEL
LIN {X 0,Y 318.541,Z 906.354,A -85,B 0,C 180,E1 -15201.755,E2 -15201.755} C_VEL
LIN {X 0,Y 318.64,Z 909.984,A -85,B 0,C 180,E1 -15203.668,E2 -15203.668} C_VEL
LIN {X 0,Y 318.774,Z 911.865,A -85,B 0,C 180,E1 -15204.94,E2 -15204.94} C_VEL
LIN {X 0,Y 318.952,Z 913.282,A -85,B 0,C 180,E1 -15206.21,E2 -15206.21} C_VEL
LIN {X 0,Y 318.997,Z 914.238,A -85,B 0,C 180,E1 -15207.474,E2 -15207.474} C_VEL
LIN {X 0,Y 319.099,Z 914.79,A -85,B 0,C 180,E1 -15208.738,E2 -15208.738} C_VEL
LIN {X 0,Y 319.244,Z 914.934,A -85,B 0,C 180,E1 -15210,E2 -15210} C_VEL
LIN {X 0,Y 319.135,Z 914.58,A -85,B 0,C 180,E1 -15211.262,E2 -15211.262} C_VEL
LIN {X 0,Y 319.06,Z 913.786,A -85,B 0,C 180,E1 -15212.525,E2 -15212.525} C_VEL
LIN {X 0,Y 318.981,Z 912.567,A -85,B 0,C 180,E1 -15213.79,E2 -15213.79} C_VEL
LIN {X 0,Y 318.835,Z 909.855,A -85,B 0,C 180,E1 -15215.693,E2 -15215.693} C_VEL
LIN {X 0,Y 318.743,Z 906.044,A -85,B 0,C 180,E1 -15217.602,E2 -15217.602} C_VEL
LIN {X 0,Y 318.752,Z 901.042,A -85,B 0,C 180,E1 -15219.518,E2 -15219.518} C_VEL
LIN {X 0,Y 319.075,Z 894.74,A -85,B 0,C 180,E1 -15221.434,E2 -15221.434} C_VEL
LIN {X 0,Y 319.772,Z 886.852,A -85,B 0,C 180,E1 -15223.342,E2 -15223.342} C_VEL
LIN {X 0,Y 320.521,Z 878.811,A -85,B 0,C 180,E1 -15224.93,E2 -15224.93} C_VEL
LIN {X 0,Y 321.627,Z 869.087,A -85,B 0,C 180,E1 -15226.503,E2 -15226.503} C_VEL
LIN {X 0,Y 322.843,Z 858.341,A -85,B 0,C 180,E1 -15227.908,E2 -15227.908} C_VEL
LIN {X 0,Y 322.45,Z 846.191,A -85,B 0,C 180,E1 -15229.207,E2 -15229.207} C_VEL
LIN {X 0,Y 321.824,Z 833.227,A -85,B 0,C 180,E1 -15230.309,E2 -15230.309} C_VEL
LIN {X 0,Y 320.729,Z 819.404,A -85,B 0,C 180,E1 -15231.196,E2 -15231.196} C_VEL
LIN {X 0,Y 319.487,Z 806.093,A -85,B 0,C 180,E1 -15231.833,E2 -15231.833} C_VEL
LIN {X 0,Y 320.611,Z 792.53,A -85,B 0,C 180,E1 -15236.703,E2 -15236.703} C_VEL
LIN {X 0,Y 321.834,Z 781.054,A -85,B 0,C 180,E1 -15240.876,E2 -15240.876} C_VEL
LIN {X 0,Y 323.389,Z 769.465,A -85,B 0,C 180,E1 -15245.163,E2 -15245.163} C_VEL
LIN {X 0,Y 324.432,Z 761.944,A -85,B 0,C 180,E1 -15248.004,E2 -15248.004} C_VEL
LIN {X 0,Y 323.292,Z 755.336,A -85,B 0,C 180,E1 -15250.705,E2 -15250.705} C_VEL
LIN {X 0,Y 321.564,Z 746.78,A -85,B 0,C 180,E1 -15254.378,E2 -15254.378} C_VEL
LIN {X 0,Y 319.843,Z 738.075,A -85,B 0,C 180,E1 -15258.339,E2 -15258.339} C_VEL
LIN {X 0,Y 319.562,Z 736.679,A -85,B 0,C 180,E1 -15259.031,E2 -15259.031} C_VEL
LIN {X 0,Y 319.563,Z 736.676,A -85,B 0,C 180,E1 -15262.348,E2 -15262.348} C_VEL
LIN {X 0,Y 319.561,Z 736.676,A -85,B 0,C 180,E1 -15265.124,E2 -15265.124} C_VEL
LIN {X 0,Y 319.571,Z 736.674,A -85,B 0,C 180,E1 -15269.058,E2 -15269.058} C_VEL
LIN {X 0,Y 319.61,Z 736.67,A -85,B 0,C 180,E1 -15272.498,E2 -15272.498} C_VEL
LIN {X 0,Y 319.605,Z 736.671,A -85,B 0,C 180,E1 -15275.304,E2 -15275.304} C_VEL
LIN {X 0,Y 319.606,Z 736.67,A -85,B 0,C 180,E1 -15279.401,E2 -15279.401} C_VEL
LIN {X 0,Y 319.66,Z 736.668,A -85,B 0,C 180,E1 -15282.073,E2 -15282.073} C_VEL
LIN {X 0,Y 319.734,Z 736.657,A -85,B 0,C 180,E1 -15286.008,E2 -15286.008} C_VEL
LIN {X 0,Y 319.754,Z 736.653,A -85,B 0,C 180,E1 -15289.873,E2 -15289.873} C_VEL
LIN {X 0,Y 319.914,Z 736.637,A -85,B 0,C 180,E1 -15292.426,E2 -15292.426} C_VEL
LIN {X 0,Y 319.739,Z 736.655,A -85,B 0,C 180,E1 -15294.956,E2 -15294.956} C_VEL
LIN {X 0,Y 319.98,Z 736.623,A -85,B 0,C 180,E1 -15297.482,E2 -15297.482} C_VEL
LIN {X 0,Y 320.114,Z 736.607,A -85,B 0,C 180,E1 -15300,E2 -15300} C_VEL
LIN {X 0,Y 319.987,Z 736.626,A -85,B 0,C 180,E1 -15302.518,E2 -15302.518} C_VEL
LIN {X 0,Y 319.893,Z 736.634,A -85,B 0,C 180,E1 -15306.491,E2 -15306.491} C_VEL
LIN {X 0,Y 319.737,Z 736.654,A -85,B 0,C 180,E1 -15310.128,E2 -15310.128} C_VEL
LIN {X 0,Y 319.734,Z 736.654,A -85,B 0,C 180,E1 -15313.992,E2 -15313.992} C_VEL
LIN {X 0,Y 319.626,Z 736.668,A -85,B 0,C 180,E1 -15317.929,E2 -15317.929} C_VEL
LIN {X 0,Y 319.566,Z 736.675,A -85,B 0,C 180,E1 -15321.955,E2 -15321.955} C_VEL
LIN {X 0,Y 319.554,Z 736.677,A -85,B 0,C 180,E1 -15326.095,E2 -15326.095} C_VEL
LIN {X 0,Y 319.545,Z 736.679,A -85,B 0,C 180,E1 -15328.938,E2 -15328.938} C_VEL
LIN {X 0,Y 319.526,Z 736.683,A -85,B 0,C 180,E1 -15331.863,E2 -15331.863} C_VEL
LIN {X 0,Y 319.58,Z 736.678,A -85,B 0,C 180,E1 -15335.543,E2 -15335.543} C_VEL
LIN {X 0,Y 319.529,Z 736.684,A -85,B 0,C 180,E1 -15339.662,E2 -15339.662} C_VEL
LIN {X 0,Y 319.52,Z 736.683,A -85,B 0,C 180,E1 -15343.46,E2 -15343.46} C_VEL
LIN {X 0,Y 319.552,Z 736.677,A -85,B 0,C 180,E1 -15347.016,E2 -15347.016} C_VEL
LIN {X 0,Y 319.515,Z 736.684,A -85,B 0,C 180,E1 -15350.366,E2 -15350.366} C_VEL
LIN {X 0,Y 319.579,Z 736.676,A -85,B 0,C 180,E1 -15354.458,E2 -15354.458} C_VEL
LIN {X 0,Y 319.525,Z 736.685,A -85,B 0,C 180,E1 -15358.137,E2 -15358.137} C_VEL
LIN {X 0,Y 319.546,Z 736.678,A -85,B 0,C 180,E1 -15361.613,E2 -15361.613} C_VEL
LIN {X 0,Y 319.528,Z 736.68,A -85,B 0,C 180,E1 -15365.298,E2 -15365.298} C_VEL
LIN {X 0,Y 319.567,Z 736.676,A -85,B 0,C 180,E1 -15368.046,E2 -15368.046} C_VEL
LIN {X 0,Y 319.627,Z 736.668,A -85,B 0,C 180,E1 -15372.071,E2 -15372.071} C_VEL
LIN {X 0,Y 319.734,Z 736.654,A -85,B 0,C 180,E1 -15376.008,E2 -15376.008} C_VEL
LIN {X 0,Y 319.736,Z 736.654,A -85,B 0,C 180,E1 -15379.872,E2 -15379.872} C_VEL
LIN {X 0,Y 319.9,Z 736.634,A -85,B 0,C 180,E1 -15383.694,E2 -15383.694} C_VEL
LIN {X 0,Y 319.956,Z 736.629,A -85,B 0,C 180,E1 -15387.482,E2 -15387.482} C_VEL
LIN {X 0,Y 320.001,Z 736.626,A -85,B 0,C 180,E1 -15391.259,E2 -15391.259} C_VEL
LIN {X 0,Y 319.706,Z 736.659,A -85,B 0,C 180,E1 -15393.781,E2 -15393.781} C_VEL
LIN {X 0,Y 319.903,Z 736.633,A -85,B 0,C 180,E1 -15396.307,E2 -15396.307} C_VEL
LIN {X 0,Y 319.738,Z 736.654,A -85,B 0,C 180,E1 -15400.128,E2 -15400.128} C_VEL
LIN {X 0,Y 319.736,Z 736.656,A -85,B 0,C 180,E1 -15403.992,E2 -15403.992} C_VEL
LIN {X 0,Y 319.662,Z 736.666,A -85,B 0,C 180,E1 -15407.927,E2 -15407.927} C_VEL
LIN {X 0,Y 319.602,Z 736.67,A -85,B 0,C 180,E1 -15410.6,E2 -15410.6} C_VEL
LIN {X 0,Y 319.576,Z 736.674,A -85,B 0,C 180,E1 -15414.699,E2 -15414.699} C_VEL
LIN {X 0,Y 319.574,Z 736.676,A -85,B 0,C 180,E1 -15418.397,E2 -15418.397} C_VEL
LIN {X 0,Y 319.527,Z 736.684,A -85,B 0,C 180,E1 -15421.863,E2 -15421.863} C_VEL
LIN {X 0,Y 319.583,Z 736.674,A -85,B 0,C 180,E1 -15425.543,E2 -15425.543} C_VEL
LIN {X 0,Y 319.576,Z 736.678,A -85,B 0,C 180,E1 -15428.008,E2 -15428.008} C_VEL
LIN {X 0,Y 319.566,Z 736.682,A -85,B 0,C 180,E1 -15431.829,E2 -15431.829} C_VEL
LIN {X 0,Y 323.337,Z 749.467,A -85,B 0,C 180,E1 -15433.043,E2 -15433.043} C_VEL
LIN {X 0,Y 325.644,Z 757.871,A -85,B 0,C 180,E1 -15433.998,E2 -15433.998} C_VEL
LIN {X 0,Y 325.642,Z 761.56,A -85,B 0,C 180,E1 -15434.407,E2 -15434.407} C_VEL
LIN {X 0,Y 324.638,Z 773.254,A -85,B 0,C 180,E1 -15435.847,E2 -15435.847} C_VEL
LIN {X 0,Y 323.743,Z 782.872,A -85,B 0,C 180,E1 -15437.324,E2 -15437.324} C_VEL
LIN {X 0,Y 322.685,Z 792.841,A -85,B 0,C 180,E1 -15439.202,E2 -15439.202} C_VEL
LIN {X 0,Y 321.861,Z 800.711,A -85,B 0,C 180,E1 -15441.053,E2 -15441.053} C_VEL
LIN {X 0,Y 321.151,Z 807.368,A -85,B 0,C 180,E1 -15443,E2 -15443} C_VEL
LIN {X 0,Y 320.508,Z 813.381,A -85,B 0,C 180,E1 -15445.241,E2 -15445.241} C_VEL
LIN {X 0,Y 320.181,Z 817.731,A -85,B 0,C 180,E1 -15447.467,E2 -15447.467} C_VEL
LIN {X 0,Y 319.95,Z 820.685,A -85,B 0,C 180,E1 -15449.654,E2 -15449.654} C_VEL
LIN {X 0,Y 319.985,Z 822.171,A -85,B 0,C 180,E1 -15451.468,E2 -15451.468} C_VEL
LIN {X 0,Y 320.22,Z 822.884,A -85,B 0,C 180,E1 -15453.963,E2 -15453.963} C_VEL
LIN {X 0,Y 320.482,Z 822.554,A -85,B 0,C 180,E1 -15455.376,E2 -15455.376} C_VEL
LIN {X 0,Y 321.096,Z 821.019,A -85,B 0,C 180,E1 -15457.57,E2 -15457.57} C_VEL
LIN {X 0,Y 321.946,Z 818.203,A -85,B 0,C 180,E1 -15459.832,E2 -15459.832} C_VEL
LIN {X 0,Y 322.749,Z 814.933,A -85,B 0,C 180,E1 -15461.594,E2 -15461.594} C_VEL
LIN {X 0,Y 323.4,Z 812.19,A -85,B 0,C 180,E1 -15462.767,E2 -15462.767} C_VEL
LIN {X 0,Y 323.321,Z 809.873,A -85,B 0,C 180,E1 -15463.732,E2 -15463.732} C_VEL
LIN {X 0,Y 321.595,Z 805.943,A -85,B 0,C 180,E1 -15465.324,E2 -15465.324} C_VEL
LIN {X 0,Y 320.02,Z 801.353,A -85,B 0,C 180,E1 -15466.865,E2 -15466.865} C_VEL
LIN {X 0,Y 320.156,Z 797.994,A -85,B 0,C 180,E1 -15467.732,E2 -15467.732} C_VEL
LIN {X 0,Y 321.726,Z 789.788,A -85,B 0,C 180,E1 -15469.425,E2 -15469.425} C_VEL
LIN {X 0,Y 323.254,Z 780.863,A -85,B 0,C 180,E1 -15470.931,E2 -15470.931} C_VEL
LIN {X 0,Y 324.788,Z 770.142,A -85,B 0,C 180,E1 -15472.384,E2 -15472.384} C_VEL
LIN {X 0,Y 323.335,Z 763.538,A -85,B 0,C 180,E1 -15473.402,E2 -15473.402} C_VEL
LIN {X 0,Y 319.751,Z 753.01,A -85,B 0,C 180,E1 -15474.956,E2 -15474.956} C_VEL
LIN {X 0,Y 314.821,Z 742.481,A -85,B 0,C 180,E1 -15476.48,E2 -15476.48} C_VEL
LIN {X 0,Y 312.959,Z 738.203,A -85,B 0,C 180,E1 -15477.023,E2 -15477.023} C_VEL
LIN {X 0,Y 312.845,Z 737.519,A -85,B 0,C 180,E1 -15477.103,E2 -15477.103} C_VEL
LIN {X 0,Y 313.07,Z 737.489,A -85,B 0,C 180,E1 -15480,E2 -15480} C_VEL
LIN {X 0,Y 312.936,Z 737.498,A -85,B 0,C 180,E1 -15482.574,E2 -15482.574} C_VEL
LIN {X 0,Y 312.902,Z 737.503,A -85,B 0,C 180,E1 -15486.448,E2 -15486.448} C_VEL
LIN {X 0,Y 312.77,Z 737.516,A -85,B 0,C 180,E1 -15489.05,E2 -15489.05} C_VEL
LIN {X 0,Y 312.638,Z 737.539,A -85,B 0,C 180,E1 -15492.991,E2 -15492.991} C_VEL
LIN {X 0,Y 312.641,Z 737.534,A -85,B 0,C 180,E1 -15495.65,E2 -15495.65} C_VEL
LIN {X 0,Y 312.632,Z 737.542,A -85,B 0,C 180,E1 -15499.236,E2 -15499.236} C_VEL
LIN {X 0,Y 312.529,Z 737.554,A -85,B 0,C 180,E1 -15502.78,E2 -15502.78} C_VEL
LIN {X 0,Y 312.599,Z 737.543,A -85,B 0,C 180,E1 -15505.933,E2 -15505.933} C_VEL
LIN {X 0,Y 312.541,Z 737.553,A -85,B 0,C 180,E1 -15509.65,E2 -15509.65} C_VEL
LIN {X 0,Y 312.522,Z 737.555,A -85,B 0,C 180,E1 -15513.689,E2 -15513.689} C_VEL
LIN {X 0,Y 312.538,Z 737.674,A -85,B 0,C 180,E1 -15515.95,E2 -15515.95} C_VEL
LIN {X 0,Y 313.577,Z 742.33,A -85,B 0,C 180,E1 -15519.649,E2 -15519.649} C_VEL
LIN {X 0,Y 314.651,Z 747.312,A -85,B 0,C 180,E1 -15523.02,E2 -15523.02} C_VEL
LIN {X 0,Y 315.77,Z 753.007,A -85,B 0,C 180,E1 -15526.373,E2 -15526.373} C_VEL
LIN {X 0,Y 317.113,Z 759.953,A -85,B 0,C 180,E1 -15530.005,E2 -15530.005} C_VEL
LIN {X 0,Y 317.484,Z 763.517,A -85,B 0,C 180,E1 -15531.696,E2 -15531.696} C_VEL
LIN {X 0,Y 316.624,Z 768.849,A -85,B 0,C 180,E1 -15533.969,E2 -15533.969} C_VEL
LIN {X 0,Y 315.38,Z 776.117,A -85,B 0,C 180,E1 -15536.909,E2 -15536.909} C_VEL
LIN {X 0,Y 314.118,Z 786.015,A -85,B 0,C 180,E1 -15540.76,E2 -15540.76} C_VEL
LIN {X 0,Y 313.102,Z 795.863,A -85,B 0,C 180,E1 -15544.439,E2 -15544.439} C_VEL
LIN {X 0,Y 316.323,Z 812.194,A -85,B 0,C 180,E1 -15545.634,E2 -15545.634} C_VEL
LIN {X 0,Y 317.871,Z 825.646,A -85,B 0,C 180,E1 -15546.745,E2 -15546.745} C_VEL
LIN {X 0,Y 318.279,Z 836.76,A -85,B 0,C 180,E1 -15547.789,E2 -15547.789} C_VEL
LIN {X 0,Y 317.87,Z 848.392,A -85,B 0,C 180,E1 -15549.044,E2 -15549.044} C_VEL
LIN {X 0,Y 317.232,Z 860.355,A -85,B 0,C 180,E1 -15550.591,E2 -15550.591} C_VEL
LIN {X 0,Y 316.653,Z 865.8,A -85,B 0,C 180,E1 -15551.394,E2 -15551.394} C_VEL
LIN {X 0,Y 314.753,Z 876.041,A -85,B 0,C 180,E1 -15553.126,E2 -15553.126} C_VEL
LIN {X 0,Y 313.353,Z 885.733,A -85,B 0,C 180,E1 -15555.161,E2 -15555.161} C_VEL
LIN {X 0,Y 312.299,Z 893.947,A -85,B 0,C 180,E1 -15557.325,E2 -15557.325} C_VEL
LIN {X 0,Y 311.641,Z 900.847,A -85,B 0,C 180,E1 -15559.606,E2 -15559.606} C_VEL
LIN {X 0,Y 311.473,Z 905.485,A -85,B 0,C 180,E1 -15561.566,E2 -15561.566} C_VEL
LIN {X 0,Y 311.548,Z 909.056,A -85,B 0,C 180,E1 -15563.524,E2 -15563.524} C_VEL
LIN {X 0,Y 311.689,Z 910.904,A -85,B 0,C 180,E1 -15564.825,E2 -15564.825} C_VEL
LIN {X 0,Y 311.905,Z 912.285,A -85,B 0,C 180,E1 -15566.124,E2 -15566.124} C_VEL
LIN {X 0,Y 311.954,Z 913.225,A -85,B 0,C 180,E1 -15567.417,E2 -15567.417} C_VEL
LIN {X 0,Y 312.065,Z 913.759,A -85,B 0,C 180,E1 -15568.709,E2 -15568.709} C_VEL
LIN {X 0,Y 312.24,Z 913.879,A -85,B 0,C 180,E1 -15570,E2 -15570} C_VEL
LIN {X 0,Y 312.11,Z 913.48,A -85,B 0,C 180,E1 -15571.29,E2 -15571.29} C_VEL
LIN {X 0,Y 312.027,Z 912.665,A -85,B 0,C 180,E1 -15572.582,E2 -15572.582} C_VEL
LIN {X 0,Y 311.94,Z 911.422,A -85,B 0,C 180,E1 -15573.875,E2 -15573.875} C_VEL
LIN {X 0,Y 311.793,Z 908.656,A -85,B 0,C 180,E1 -15575.822,E2 -15575.822} C_VEL
LIN {X 0,Y 311.684,Z 904.783,A -85,B 0,C 180,E1 -15577.775,E2 -15577.775} C_VEL
LIN {X 0,Y 311.724,Z 899.721,A -85,B 0,C 180,E1 -15579.735,E2 -15579.735} C_VEL
LIN {X 0,Y 312.067,Z 893.326,A -85,B 0,C 180,E1 -15581.694,E2 -15581.694} C_VEL
LIN {X 0,Y 312.836,Z 885.343,A -85,B 0,C 180,E1 -15583.644,E2 -15583.644} C_VEL
LIN {X 0,Y 313.728,Z 876.395,A -85,B 0,C 180,E1 -15585.414,E2 -15585.414} C_VEL
LIN {X 0,Y 314.876,Z 866.257,A -85,B 0,C 180,E1 -15587.035,E2 -15587.035} C_VEL
LIN {X 0,Y 315.79,Z 857.753,A -85,B 0,C 180,E1 -15588.154,E2 -15588.154} C_VEL
LIN {X 0,Y 315.454,Z 847.047,A -85,B 0,C 180,E1 -15589.354,E2 -15589.354} C_VEL
LIN {X 0,Y 314.855,Z 833.723,A -85,B 0,C 180,E1 -15590.547,E2 -15590.547} C_VEL
LIN {X 0,Y 313.917,Z 820.799,A -85,B 0,C 180,E1 -15591.442,E2 -15591.442} C_VEL
LIN {X 0,Y 312.524,Z 806.501,A -85,B 0,C 180,E1 -15592.144,E2 -15592.144} C_VEL
LIN {X 0,Y 312.448,Z 805.194,A -85,B 0,C 180,E1 -15592.22,E2 -15592.22} C_VEL
LIN {X 0,Y 313.491,Z 793.182,A -85,B 0,C 180,E1 -15596.639,E2 -15596.639} C_VEL
LIN {X 0,Y 314.747,Z 781.755,A -85,B 0,C 180,E1 -15600.902,E2 -15600.902} C_VEL
LIN {X 0,Y 316.166,Z 771.795,A -85,B 0,C 180,E1 -15604.667,E2 -15604.667} C_VEL
LIN {X 0,Y 317.321,Z 764.1,A -85,B 0,C 180,E1 -15607.621,E2 -15607.621} C_VEL
LIN {X 0,Y 317.045,Z 760.439,A -85,B 0,C 180,E1 -15609.118,E2 -15609.118} C_VEL
LIN {X 0,Y 315.426,Z 752.145,A -85,B 0,C 180,E1 -15612.67,E2 -15612.67} C_VEL
LIN {X 0,Y 313.88,Z 744.648,A -85,B 0,C 180,E1 -15616.043,E2 -15616.043} C_VEL
LIN {X 0,Y 312.53,Z 737.557,A -85,B 0,C 180,E1 -15619.469,E2 -15619.469} C_VEL
LIN {X 0,Y 312.527,Z 737.552,A -85,B 0,C 180,E1 -15622.615,E2 -15622.615} C_VEL
LIN {X 0,Y 312.521,Z 737.554,A -85,B 0,C 180,E1 -15626.311,E2 -15626.311} C_VEL
LIN {X 0,Y 312.546,Z 737.551,A -85,B 0,C 180,E1 -15630.35,E2 -15630.35} C_VEL
LIN {X 0,Y 312.604,Z 737.547,A -85,B 0,C 180,E1 -15634.064,E2 -15634.064} C_VEL
LIN {X 0,Y 312.567,Z 737.548,A -85,B 0,C 180,E1 -15637.527,E2 -15637.527} C_VEL
LIN {X 0,Y 312.64,Z 737.539,A -85,B 0,C 180,E1 -15641.657,E2 -15641.657} C_VEL
LIN {X 0,Y 312.695,Z 737.532,A -85,B 0,C 180,E1 -15645.686,E2 -15645.686} C_VEL
LIN {X 0,Y 312.7,Z 737.53,A -85,B 0,C 180,E1 -15649.642,E2 -15649.642} C_VEL
LIN {X 0,Y 312.855,Z 737.515,A -85,B 0,C 180,E1 -15652.254,E2 -15652.254} C_VEL
LIN {X 0,Y 312.902,Z 737.505,A -85,B 0,C 180,E1 -15653.552,E2 -15653.552} C_VEL
LIN {X 0,Y 312.987,Z 737.499,A -85,B 0,C 180,E1 -15658.713,E2 -15658.713} C_VEL
LIN {X 0,Y 312.986,Z 737.496,A -85,B 0,C 180,E1 -15661.287,E2 -15661.287} C_VEL
LIN {X 0,Y 312.704,Z 737.532,A -85,B 0,C 180,E1 -15665.158,E2 -15665.158} C_VEL
LIN {X 0,Y 312.804,Z 737.517,A -85,B 0,C 180,E1 -15667.748,E2 -15667.748} C_VEL
LIN {X 0,Y 312.666,Z 737.535,A -85,B 0,C 180,E1 -15671.672,E2 -15671.672} C_VEL
LIN {X 0,Y 312.669,Z 737.538,A -85,B 0,C 180,E1 -15674.865,E2 -15674.865} C_VEL
LIN {X 0,Y 312.587,Z 737.55,A -85,B 0,C 180,E1 -15679.213,E2 -15679.213} C_VEL
LIN {X 0,Y 312.515,Z 737.555,A -85,B 0,C 180,E1 -15682.775,E2 -15682.775} C_VEL
LIN {X 0,Y 312.488,Z 737.557,A -85,B 0,C 180,E1 -15686.732,E2 -15686.732} C_VEL
LIN {X 0,Y 312.498,Z 737.56,A -85,B 0,C 180,E1 -15689.655,E2 -15689.655} C_VEL
LIN {X 0,Y 312.521,Z 737.557,A -85,B 0,C 180,E1 -15693.689,E2 -15693.689} C_VEL
LIN {X 0,Y 312.512,Z 737.557,A -85,B 0,C 180,E1 -15697.387,E2 -15697.387} C_VEL
LIN {X 0,Y 312.441,Z 737.562,A -85,B 0,C 180,E1 -15700.717,E2 -15700.717} C_VEL
LIN {X 0,Y 312.451,Z 737.564,A -85,B 0,C 180,E1 -15704.21,E2 -15704.21} C_VEL
LIN {X 0,Y 312.456,Z 737.566,A -85,B 0,C 180,E1 -15707.925,E2 -15707.925} C_VEL
LIN {X 0,Y 312.477,Z 737.562,A -85,B 0,C 180,E1 -15711.925,E2 -15711.925} C_VEL
LIN {X 0,Y 312.531,Z 737.557,A -85,B 0,C 180,E1 -15714.22,E2 -15714.22} C_VEL
LIN {X 0,Y 312.503,Z 737.555,A -85,B 0,C 180,E1 -15717.334,E2 -15717.334} C_VEL
LIN {X 0,Y 312.486,Z 737.557,A -85,B 0,C 180,E1 -15721.299,E2 -15721.299} C_VEL
LIN {X 0,Y 312.518,Z 737.556,A -85,B 0,C 180,E1 -15724.705,E2 -15724.705} C_VEL
LIN {X 0,Y 312.541,Z 737.55,A -85,B 0,C 180,E1 -15727.525,E2 -15727.525} C_VEL
LIN {X 0,Y 312.585,Z 737.544,A -85,B 0,C 180,E1 -15731.653,E2 -15731.653} C_VEL
LIN {X 0,Y 312.688,Z 737.531,A -85,B 0,C 180,E1 -15735.686,E2 -15735.686} C_VEL
LIN {X 0,Y 312.686,Z 737.532,A -85,B 0,C 180,E1 -15739.641,E2 -15739.641} C_VEL
LIN {X 0,Y 312.798,Z 737.519,A -85,B 0,C 180,E1 -15742.253,E2 -15742.253} C_VEL
LIN {X 0,Y 312.688,Z 737.536,A -85,B 0,C 180,E1 -15744.842,E2 -15744.842} C_VEL
LIN {X 0,Y 312.978,Z 737.498,A -85,B 0,C 180,E1 -15748.713,E2 -15748.713} C_VEL
LIN {X 0,Y 312.907,Z 737.505,A -85,B 0,C 180,E1 -15752.575,E2 -15752.575} C_VEL
LIN {X 0,Y 312.844,Z 737.512,A -85,B 0,C 180,E1 -15756.449,E2 -15756.449} C_VEL
LIN {X 0,Y 312.754,Z 737.526,A -85,B 0,C 180,E1 -15759.05,E2 -15759.05} C_VEL
LIN {X 0,Y 312.637,Z 737.539,A -85,B 0,C 180,E1 -15762.991,E2 -15762.991} C_VEL
LIN {X 0,Y 312.642,Z 737.543,A -85,B 0,C 180,E1 -15765.65,E2 -15765.65} C_VEL
LIN {X 0,Y 312.612,Z 737.543,A -85,B 0,C 180,E1 -15769.225,E2 -15769.225} C_VEL
LIN {X 0,Y 312.524,Z 737.552,A -85,B 0,C 180,E1 -15772.778,E2 -15772.778} C_VEL
LIN {X 0,Y 312.533,Z 737.557,A -85,B 0,C 180,E1 -15775.908,E2 -15775.908} C_VEL
LIN {X 0,Y 312.499,Z 737.558,A -85,B 0,C 180,E1 -15779.655,E2 -15779.655} C_VEL
LIN {X 0,Y 312.522,Z 737.555,A -85,B 0,C 180,E1 -15783.689,E2 -15783.689} C_VEL
LIN {X 0,Y 312.528,Z 737.552,A -85,B 0,C 180,E1 -15787.385,E2 -15787.385} C_VEL
LIN {X 0,Y 312.522,Z 737.565,A -85,B 0,C 180,E1 -15791.479,E2 -15791.479} C_VEL
LIN {X 0,Y 315.777,Z 748.567,A -85,B 0,C 180,E1 -15792.528,E2 -15792.528} C_VEL
LIN {X 0,Y 318.746,Z 759.416,A -85,B 0,C 180,E1 -15793.772,E2 -15793.772} C_VEL
LIN {X 0,Y 318.67,Z 763.6,A -85,B 0,C 180,E1 -15794.249,E2 -15794.249} C_VEL
LIN {X 0,Y 317.736,Z 774.305,A -85,B 0,C 180,E1 -15795.612,E2 -15795.612} C_VEL
LIN {X 0,Y 316.788,Z 784.182,A -85,B 0,C 180,E1 -15797.166,E2 -15797.166} C_VEL
LIN {X 0,Y 315.826,Z 792.775,A -85,B 0,C 180,E1 -15798.804,E2 -15798.804} C_VEL
LIN {X 0,Y 315.025,Z 800.191,A -85,B 0,C 180,E1 -15800.519,E2 -15800.519} C_VEL
LIN {X 0,Y 314.298,Z 807.128,A -85,B 0,C 180,E1 -15802.489,E2 -15802.489} C_VEL
LIN {X 0,Y 313.694,Z 812.434,A -85,B 0,C 180,E1 -15804.373,E2 -15804.373} C_VEL
LIN {X 0,Y 313.286,Z 817.513,A -85,B 0,C 180,E1 -15806.747,E2 -15806.747} C_VEL
LIN {X 0,Y 313.009,Z 820.824,A -85,B 0,C 180,E1 -15808.907,E2 -15808.907} C_VEL
LIN {X 0,Y 312.95,Z 823.004,A -85,B 0,C 180,E1 -15811.145,E2 -15811.145} C_VEL
LIN {X 0,Y 313.197,Z 823.958,A -85,B 0,C 180,E1 -15813.843,E2 -15813.843} C_VEL
LIN {X 0,Y 313.696,Z 823.379,A -85,B 0,C 180,E1 -15816.217,E2 -15816.217} C_VEL
LIN {X 0,Y 314.152,Z 822.318,A -85,B 0,C 180,E1 -15817.647,E2 -15817.647} C_VEL
LIN {X 0,Y 314.907,Z 820.05,A -85,B 0,C 180,E1 -15819.611,E2 -15819.611} C_VEL
LIN {X 0,Y 315.934,Z 816.211,A -85,B 0,C 180,E1 -15821.854,E2 -15821.854} C_VEL
LIN {X 0,Y 317.189,Z 811.318,A -85,B 0,C 180,E1 -15823.921,E2 -15823.921} C_VEL
LIN {X 0,Y 318.712,Z 804.835,A -85,B 0,C 180,E1 -15825.992,E2 -15825.992} C_VEL
LIN {X 0,Y 320.156,Z 797.994,A -85,B 0,C 180,E1 -15827.732,E2 -15827.732} C_VEL
LIN {X 0,Y 320.309,Z 794.454,A -85,B 0,C 180,E1 -15828.581,E2 -15828.581} C_VEL
LIN {X 0,Y 318.871,Z 788.725,A -85,B 0,C 180,E1 -15830.016,E2 -15830.016} C_VEL
LIN {X 0,Y 317.454,Z 782.44,A -85,B 0,C 180,E1 -15831.368,E2 -15831.368} C_VEL
LIN {X 0,Y 317.602,Z 778.042,A -85,B 0,C 180,E1 -15832.073,E2 -15832.073} C_VEL
LIN {X 0,Y 318.494,Z 772.028,A -85,B 0,C 180,E1 -15832.87,E2 -15832.87} C_VEL
LIN {X 0,Y 316.243,Z 763.042,A -85,B 0,C 180,E1 -15834.327,E2 -15834.327} C_VEL
LIN {X 0,Y 312.896,Z 753.816,A -85,B 0,C 180,E1 -15835.765,E2 -15835.765} C_VEL
LIN {X 0,Y 307.938,Z 743.153,A -85,B 0,C 180,E1 -15837.384,E2 -15837.384} C_VEL
LIN {X 0,Y 306.035,Z 739.164,A -85,B 0,C 180,E1 -15837.944,E2 -15837.944} C_VEL
LIN {X 0,Y 305.905,Z 738.383,A -85,B 0,C 180,E1 -15838.025,E2 -15838.025} C_VEL
LIN {X 0,Y 306.026,Z 738.367,A -85,B 0,C 180,E1 -15840,E2 -15840} C_VEL
LIN {X 0,Y 305.885,Z 738.376,A -85,B 0,C 180,E1 -15842.634,E2 -15842.634} C_VEL
LIN {X 0,Y 305.844,Z 738.383,A -85,B 0,C 180,E1 -15846.597,E2 -15846.597} C_VEL
LIN {X 0,Y 305.707,Z 738.396,A -85,B 0,C 180,E1 -15849.261,E2 -15849.261} C_VEL
LIN {X 0,Y 305.592,Z 738.418,A -85,B 0,C 180,E1 -15853.296,E2 -15853.296} C_VEL
LIN {X 0,Y 305.597,Z 738.414,A -85,B 0,C 180,E1 -15856.02,E2 -15856.02} C_VEL
LIN {X 0,Y 305.578,Z 738.421,A -85,B 0,C 180,E1 -15859.444,E2 -15859.444} C_VEL
LIN {X 0,Y 305.488,Z 738.43,A -85,B 0,C 180,E1 -15863.039,E2 -15863.039} C_VEL
LIN {X 0,Y 305.528,Z 738.422,A -85,B 0,C 180,E1 -15866.219,E2 -15866.219} C_VEL
LIN {X 0,Y 305.49,Z 738.428,A -85,B 0,C 180,E1 -15869.047,E2 -15869.047} C_VEL
LIN {X 0,Y 305.445,Z 738.438,A -85,B 0,C 180,E1 -15871.952,E2 -15871.952} C_VEL
LIN {X 0,Y 305.49,Z 738.565,A -85,B 0,C 180,E1 -15874.677,E2 -15874.677} C_VEL
LIN {X 0,Y 306.435,Z 742.692,A -85,B 0,C 180,E1 -15878.26,E2 -15878.26} C_VEL
LIN {X 0,Y 307.644,Z 748.292,A -85,B 0,C 180,E1 -15882.299,E2 -15882.299} C_VEL
LIN {X 0,Y 308.776,Z 753.957,A -85,B 0,C 180,E1 -15885.804,E2 -15885.804} C_VEL
LIN {X 0,Y 310.133,Z 761.143,A -85,B 0,C 180,E1 -15889.705,E2 -15889.705} C_VEL
LIN {X 0,Y 310.56,Z 764.814,A -85,B 0,C 180,E1 -15891.513,E2 -15891.513} C_VEL
LIN {X 0,Y 309.691,Z 770.159,A -85,B 0,C 180,E1 -15893.84,E2 -15893.84} C_VEL
LIN {X 0,Y 308.092,Z 779.165,A -85,B 0,C 180,E1 -15897.567,E2 -15897.567} C_VEL
LIN {X 0,Y 306.901,Z 788.465,A -85,B 0,C 180,E1 -15901.256,E2 -15901.256} C_VEL
LIN {X 0,Y 306.276,Z 794.462,A -85,B 0,C 180,E1 -15903.567,E2 -15903.567} C_VEL
LIN {X 0,Y 308.024,Z 802.311,A -85,B 0,C 180,E1 -15904.152,E2 -15904.152} C_VEL
LIN {X 0,Y 310.512,Z 816.739,A -85,B 0,C 180,E1 -15905.341,E2 -15905.341} C_VEL
LIN {X 0,Y 311.644,Z 830.223,A -85,B 0,C 180,E1 -15906.58,E2 -15906.58} C_VEL
LIN {X 0,Y 311.526,Z 843.536,A -85,B 0,C 180,E1 -15907.974,E2 -15907.974} C_VEL
LIN {X 0,Y 310.7,Z 855.545,A -85,B 0,C 180,E1 -15909.475,E2 -15909.475} C_VEL
LIN {X 0,Y 310.114,Z 864.478,A -85,B 0,C 180,E1 -15910.815,E2 -15910.815} C_VEL
LIN {X 0,Y 308.255,Z 873.903,A -85,B 0,C 180,E1 -15912.417,E2 -15912.417} C_VEL
LIN {X 0,Y 306.8,Z 882.412,A -85,B 0,C 180,E1 -15914.178,E2 -15914.178} C_VEL
LIN {X 0,Y 305.729,Z 889.805,A -85,B 0,C 180,E1 -15916.032,E2 -15916.032} C_VEL
LIN {X 0,Y 304.931,Z 896.344,A -85,B 0,C 180,E1 -15918.028,E2 -15918.028} C_VEL
LIN {X 0,Y 304.492,Z 901.656,A -85,B 0,C 180,E1 -15920.031,E2 -15920.031} C_VEL
LIN {X 0,Y 304.378,Z 905.877,A -85,B 0,C 180,E1 -15922.037,E2 -15922.037} C_VEL
LIN {X 0,Y 304.476,Z 908.14,A -85,B 0,C 180,E1 -15923.372,E2 -15923.372} C_VEL
LIN {X 0,Y 304.604,Z 909.933,A -85,B 0,C 180,E1 -15924.704,E2 -15924.704} C_VEL
LIN {X 0,Y 304.856,Z 911.291,A -85,B 0,C 180,E1 -15926.034,E2 -15926.034} C_VEL
LIN {X 0,Y 304.912,Z 912.209,A -85,B 0,C 180,E1 -15927.358,E2 -15927.358} C_VEL
LIN {X 0,Y 305.03,Z 912.724,A -85,B 0,C 180,E1 -15928.68,E2 -15928.68} C_VEL
LIN {X 0,Y 305.234,Z 912.799,A -85,B 0,C 180,E1 -15930,E2 -15930} C_VEL
LIN {X 0,Y 305.086,Z 912.372,A -85,B 0,C 180,E1 -15931.32,E2 -15931.32} C_VEL
LIN {X 0,Y 304.994,Z 911.533,A -85,B 0,C 180,E1 -15932.641,E2 -15932.641} C_VEL
LIN {X 0,Y 304.901,Z 910.265,A -85,B 0,C 180,E1 -15933.965,E2 -15933.965} C_VEL
LIN {X 0,Y 304.73,Z 907.442,A -85,B 0,C 180,E1 -15935.957,E2 -15935.957} C_VEL
LIN {X 0,Y 304.618,Z 903.508,A -85,B 0,C 180,E1 -15937.957,E2 -15937.957} C_VEL
LIN {X 0,Y 304.737,Z 897.367,A -85,B 0,C 180,E1 -15940.296,E2 -15940.296} C_VEL
LIN {X 0,Y 305.213,Z 890.646,A -85,B 0,C 180,E1 -15942.298,E2 -15942.298} C_VEL
LIN {X 0,Y 306,Z 882.303,A -85,B 0,C 180,E1 -15944.294,E2 -15944.294} C_VEL
LIN {X 0,Y 306.951,Z 873.743,A -85,B 0,C 180,E1 -15945.947,E2 -15945.947} C_VEL
LIN {X 0,Y 308.213,Z 863.291,A -85,B 0,C 180,E1 -15947.586,E2 -15947.586} C_VEL
LIN {X 0,Y 308.714,Z 857.092,A -85,B 0,C 180,E1 -15948.413,E2 -15948.413} C_VEL
LIN {X 0,Y 308.441,Z 846.457,A -85,B 0,C 180,E1 -15949.639,E2 -15949.639} C_VEL
LIN {X 0,Y 307.891,Z 833.965,A -85,B 0,C 180,E1 -15950.796,E2 -15950.796} C_VEL
LIN {X 0,Y 306.931,Z 820.725,A -85,B 0,C 180,E1 -15951.756,E2 -15951.756} C_VEL
LIN {X 0,Y 305.661,Z 806.94,A -85,B 0,C 180,E1 -15952.473,E2 -15952.473} C_VEL
LIN {X 0,Y 305.429,Z 804.221,A -85,B 0,C 180,E1 -15952.625,E2 -15952.625} C_VEL
LIN {X 0,Y 306.563,Z 791.909,A -85,B 0,C 180,E1 -15957.291,E2 -15957.291} C_VEL
LIN {X 0,Y 307.669,Z 782.418,A -85,B 0,C 180,E1 -15960.928,E2 -15960.928} C_VEL
LIN {X 0,Y 309.249,Z 771.65,A -85,B 0,C 180,E1 -15965.101,E2 -15965.101} C_VEL
LIN {X 0,Y 310.329,Z 764.084,A -85,B 0,C 180,E1 -15968.107,E2 -15968.107} C_VEL
LIN {X 0,Y 309.457,Z 758.53,A -85,B 0,C 180,E1 -15970.465,E2 -15970.465} C_VEL
LIN {X 0,Y 307.868,Z 750.567,A -85,B 0,C 180,E1 -15974.021,E2 -15974.021} C_VEL
LIN {X 0,Y 306.085,Z 741.586,A -85,B 0,C 180,E1 -15978.251,E2 -15978.251} C_VEL
LIN {X 0,Y 305.479,Z 738.435,A -85,B 0,C 180,E1 -15979.896,E2 -15979.896} C_VEL
LIN {X 0,Y 305.482,Z 738.434,A -85,B 0,C 180,E1 -15983.632,E2 -15983.632} C_VEL
LIN {X 0,Y 305.466,Z 738.432,A -85,B 0,C 180,E1 -15986.483,E2 -15986.483} C_VEL
LIN {X 0,Y 305.465,Z 738.435,A -85,B 0,C 180,E1 -15989.591,E2 -15989.591} C_VEL
LIN {X 0,Y 305.522,Z 738.424,A -85,B 0,C 180,E1 -15992.609,E2 -15992.609} C_VEL
LIN {X 0,Y 305.507,Z 738.428,A -85,B 0,C 180,E1 -15995.539,E2 -15995.539} C_VEL
LIN {X 0,Y 305.514,Z 738.428,A -85,B 0,C 180,E1 -15999.815,E2 -15999.815} C_VEL
LIN {X 0,Y 305.576,Z 738.419,A -85,B 0,C 180,E1 -16002.603,E2 -16002.603} C_VEL
LIN {X 0,Y 305.651,Z 738.408,A -85,B 0,C 180,E1 -16005.349,E2 -16005.349} C_VEL
LIN {X 0,Y 305.637,Z 738.41,A -85,B 0,C 180,E1 -16009.4,E2 -16009.4} C_VEL
LIN {X 0,Y 305.798,Z 738.392,A -85,B 0,C 180,E1 -16012.074,E2 -16012.074} C_VEL
LIN {X 0,Y 305.682,Z 738.408,A -85,B 0,C 180,E1 -16014.723,E2 -16014.723} C_VEL
LIN {X 0,Y 305.954,Z 738.376,A -85,B 0,C 180,E1 -16018.684,E2 -16018.684} C_VEL
LIN {X 0,Y 305.954,Z 738.371,A -85,B 0,C 180,E1 -16021.316,E2 -16021.316} C_VEL
LIN {X 0,Y 305.673,Z 738.407,A -85,B 0,C 180,E1 -16025.277,E2 -16025.277} C_VEL
LIN {X 0,Y 305.753,Z 738.395,A -85,B 0,C 180,E1 -16027.927,E2 -16027.927} C_VEL
LIN {X 0,Y 305.601,Z 738.415,A -85,B 0,C 180,E1 -16031.945,E2 -16031.945} C_VEL
LIN {X 0,Y 305.611,Z 738.418,A -85,B 0,C 180,E1 -16035.015,E2 -16035.015} C_VEL
LIN {X 0,Y 305.544,Z 738.425,A -85,B 0,C 180,E1 -16039.427,E2 -16039.427} C_VEL
LIN {X 0,Y 305.456,Z 738.436,A -85,B 0,C 180,E1 -16043.026,E2 -16043.026} C_VEL
LIN {X 0,Y 305.455,Z 738.433,A -85,B 0,C 180,E1 -16046.191,E2 -16046.191} C_VEL
LIN {X 0,Y 305.45,Z 738.435,A -85,B 0,C 180,E1 -16049.034,E2 -16049.034} C_VEL
LIN {X 0,Y 305.438,Z 738.437,A -85,B 0,C 180,E1 -16051.953,E2 -16051.953} C_VEL
LIN {X 0,Y 305.462,Z 738.433,A -85,B 0,C 180,E1 -16055.114,E2 -16055.114} C_VEL
LIN {X 0,Y 305.412,Z 738.438,A -85,B 0,C 180,E1 -16058.52,E2 -16058.52} C_VEL
LIN {X 0,Y 305.436,Z 738.435,A -85,B 0,C 180,E1 -16062.582,E2 -16062.582} C_VEL
LIN {X 0,Y 305.422,Z 738.439,A -85,B 0,C 180,E1 -16066.344,E2 -16066.344} C_VEL
LIN {X 0,Y 305.411,Z 738.442,A -85,B 0,C 180,E1 -16069.885,E2 -16069.885} C_VEL
LIN {X 0,Y 305.463,Z 738.433,A -85,B 0,C 180,E1 -16073.637,E2 -16073.637} C_VEL
LIN {X 0,Y 305.466,Z 738.435,A -85,B 0,C 180,E1 -16076.483,E2 -16076.483} C_VEL
LIN {X 0,Y 305.418,Z 738.437,A -85,B 0,C 180,E1 -16079.586,E2 -16079.586} C_VEL
LIN {X 0,Y 305.443,Z 738.438,A -85,B 0,C 180,E1 -16082.601,E2 -16082.601} C_VEL
LIN {X 0,Y 305.442,Z 738.434,A -85,B 0,C 180,E1 -16085.533,E2 -16085.533} C_VEL
LIN {X 0,Y 305.498,Z 738.427,A -85,B 0,C 180,E1 -16089.814,E2 -16089.814} C_VEL
LIN {X 0,Y 305.545,Z 738.427,A -85,B 0,C 180,E1 -16092.601,E2 -16092.601} C_VEL
LIN {X 0,Y 305.629,Z 738.412,A -85,B 0,C 180,E1 -16095.348,E2 -16095.348} C_VEL
LIN {X 0,Y 305.625,Z 738.413,A -85,B 0,C 180,E1 -16099.399,E2 -16099.399} C_VEL
LIN {X 0,Y 305.748,Z 738.396,A -85,B 0,C 180,E1 -16102.073,E2 -16102.073} C_VEL
LIN {X 0,Y 305.658,Z 738.41,A -85,B 0,C 180,E1 -16104.723,E2 -16104.723} C_VEL
LIN {X 0,Y 305.946,Z 738.373,A -85,B 0,C 180,E1 -16108.684,E2 -16108.684} C_VEL
LIN {X 0,Y 305.938,Z 738.377,A -85,B 0,C 180,E1 -16111.316,E2 -16111.316} C_VEL
LIN {X 0,Y 305.662,Z 738.412,A -85,B 0,C 180,E1 -16115.277,E2 -16115.277} C_VEL
LIN {X 0,Y 305.749,Z 738.397,A -85,B 0,C 180,E1 -16117.928,E2 -16117.928} C_VEL
LIN {X 0,Y 305.602,Z 738.416,A -85,B 0,C 180,E1 -16121.945,E2 -16121.945} C_VEL
LIN {X 0,Y 305.641,Z 738.411,A -85,B 0,C 180,E1 -16125.035,E2 -16125.035} C_VEL
LIN {X 0,Y 305.583,Z 738.417,A -85,B 0,C 180,E1 -16128.783,E2 -16128.783} C_VEL
LIN {X 0,Y 305.489,Z 738.429,A -85,B 0,C 180,E1 -16133.039,E2 -16133.039} C_VEL
LIN {X 0,Y 305.473,Z 738.434,A -85,B 0,C 180,E1 -16136.197,E2 -16136.197} C_VEL
LIN {X 0,Y 305.452,Z 738.433,A -85,B 0,C 180,E1 -16139.034,E2 -16139.034} C_VEL
LIN {X 0,Y 305.439,Z 738.44,A -85,B 0,C 180,E1 -16141.953,E2 -16141.953} C_VEL
LIN {X 0,Y 305.465,Z 738.432,A -85,B 0,C 180,E1 -16145.113,E2 -16145.113} C_VEL
LIN {X 0,Y 305.47,Z 738.434,A -85,B 0,C 180,E1 -16148.533,E2 -16148.533} C_VEL
LIN {X 0,Y 305.46,Z 738.516,A -85,B 0,C 180,E1 -16151.127,E2 -16151.127} C_VEL
LIN {X 0,Y 309.277,Z 751.302,A -85,B 0,C 180,E1 -16152.398,E2 -16152.398} C_VEL
LIN {X 0,Y 312.026,Z 762.096,A -85,B 0,C 180,E1 -16153.69,E2 -16153.69} C_VEL
LIN {X 0,Y 310.981,Z 773.346,A -85,B 0,C 180,E1 -16155.095,E2 -16155.095} C_VEL
LIN {X 0,Y 309.936,Z 784.252,A -85,B 0,C 180,E1 -16156.792,E2 -16156.792} C_VEL
LIN {X 0,Y 308.822,Z 794.097,A -85,B 0,C 180,E1 -16158.702,E2 -16158.702} C_VEL
LIN {X 0,Y 307.913,Z 802.284,A -85,B 0,C 180,E1 -16160.669,E2 -16160.669} C_VEL
LIN {X 0,Y 307.195,Z 808.839,A -85,B 0,C 180,E1 -16162.635,E2 -16162.635} C_VEL
LIN {X 0,Y 306.482,Z 815.099,A -85,B 0,C 180,E1 -16165.02,E2 -16165.02} C_VEL
LIN {X 0,Y 306.151,Z 819.602,A -85,B 0,C 180,E1 -16167.352,E2 -16167.352} C_VEL
LIN {X 0,Y 305.942,Z 822.659,A -85,B 0,C 180,E1 -16169.643,E2 -16169.643} C_VEL
LIN {X 0,Y 305.941,Z 824.015,A -85,B 0,C 180,E1 -16171.157,E2 -16171.157} C_VEL
LIN {X 0,Y 306.134,Z 825.02,A -85,B 0,C 180,E1 -16173.552,E2 -16173.552} C_VEL
LIN {X 0,Y 306.745,Z 824.504,A -85,B 0,C 180,E1 -16176.415,E2 -16176.415} C_VEL
LIN {X 0,Y 307.514,Z 822.845,A -85,B 0,C 180,E1 -16178.551,E2 -16178.551} C_VEL
LIN {X 0,Y 308.354,Z 820.059,A -85,B 0,C 180,E1 -16180.702,E2 -16180.702} C_VEL
LIN {X 0,Y 309.531,Z 816.043,A -85,B 0,C 180,E1 -16182.832,E2 -16182.832} C_VEL
LIN {X 0,Y 310.958,Z 810.725,A -85,B 0,C 180,E1 -16184.935,E2 -16184.935} C_VEL
LIN {X 0,Y 312.626,Z 803.952,A -85,B 0,C 180,E1 -16187.008,E2 -16187.008} C_VEL
LIN {X 0,Y 314.355,Z 795.751,A -85,B 0,C 180,E1 -16188.983,E2 -16188.983} C_VEL
LIN {X 0,Y 316.139,Z 786.681,A -85,B 0,C 180,E1 -16190.725,E2 -16190.725} C_VEL
LIN {X 0,Y 317.602,Z 778.042,A -85,B 0,C 180,E1 -16192.073,E2 -16192.073} C_VEL
LIN {X 0,Y 317.327,Z 775.208,A -85,B 0,C 180,E1 -16192.547,E2 -16192.547} C_VEL
LIN {X 0,Y 315.974,Z 772.871,A -85,B 0,C 180,E1 -16193.074,E2 -16193.074} C_VEL
LIN {X 0,Y 310.845,Z 767.2,A -85,B 0,C 180,E1 -16194.526,E2 -16194.526} C_VEL
LIN {X 0,Y 309.974,Z 765.367,A -85,B 0,C 180,E1 -16194.871,E2 -16194.871} C_VEL
LIN {X 0,Y 306.65,Z 756.227,A -85,B 0,C 180,E1 -16196.386,E2 -16196.386} C_VEL
LIN {X 0,Y 301.181,Z 744.312,A -85,B 0,C 180,E1 -16198.295,E2 -16198.295} C_VEL
LIN {X 0,Y 299.175,Z 740.388,A -85,B 0,C 180,E1 -16198.906,E2 -16198.906} C_VEL
LIN {X 0,Y 298.933,Z 739.249,A -85,B 0,C 180,E1 -16199.074,E2 -16199.074} C_VEL
LIN {X 0,Y 298.835,Z 739.253,A -85,B 0,C 180,E1 -16202.696,E2 -16202.696} C_VEL
LIN {X 0,Y 298.789,Z 739.262,A -85,B 0,C 180,E1 -16206.754,E2 -16206.754} C_VEL
LIN {X 0,Y 298.638,Z 739.277,A -85,B 0,C 180,E1 -16209.482,E2 -16209.482} C_VEL
LIN {X 0,Y 298.556,Z 739.297,A -85,B 0,C 180,E1 -16213.615,E2 -16213.615} C_VEL
LIN {X 0,Y 298.552,Z 739.297,A -85,B 0,C 180,E1 -16216.408,E2 -16216.408} C_VEL
LIN {X 0,Y 298.512,Z 739.302,A -85,B 0,C 180,E1 -16219.654,E2 -16219.654} C_VEL
LIN {X 0,Y 298.431,Z 739.305,A -85,B 0,C 180,E1 -16223.6,E2 -16223.6} C_VEL
LIN {X 0,Y 298.488,Z 739.299,A -85,B 0,C 180,E1 -16226.575,E2 -16226.575} C_VEL
LIN {X 0,Y 298.419,Z 739.311,A -85,B 0,C 180,E1 -16229.641,E2 -16229.641} C_VEL
LIN {X 0,Y 298.412,Z 739.405,A -85,B 0,C 180,E1 -16233.2,E2 -16233.2} C_VEL
LIN {X 0,Y 299.352,Z 743.431,A -85,B 0,C 180,E1 -16237.038,E2 -16237.038} C_VEL
LIN {X 0,Y 300.449,Z 748.404,A -85,B 0,C 180,E1 -16240.917,E2 -16240.917} C_VEL
LIN {X 0,Y 301.507,Z 753.552,A -85,B 0,C 180,E1 -16244.37,E2 -16244.37} C_VEL
LIN {X 0,Y 302.638,Z 759.782,A -85,B 0,C 180,E1 -16247.998,E2 -16247.998} C_VEL
LIN {X 0,Y 303.544,Z 764.703,A -85,B 0,C 180,E1 -16250.614,E2 -16250.614} C_VEL
LIN {X 0,Y 303.517,Z 767.445,A -85,B 0,C 180,E1 -16251.932,E2 -16251.932} C_VEL
LIN {X 0,Y 302.097,Z 775.006,A -85,B 0,C 180,E1 -16255.252,E2 -16255.252} C_VEL
LIN {X 0,Y 300.263,Z 786.441,A -85,B 0,C 180,E1 -16260,E2 -16260} C_VEL
LIN {X 0,Y 299.514,Z 792.923,A -85,B 0,C 180,E1 -16262.585,E2 -16262.585} C_VEL
LIN {X 0,Y 300.401,Z 797.055,A -85,B 0,C 180,E1 -16262.926,E2 -16262.926} C_VEL
LIN {X 0,Y 303.249,Z 811.238,A -85,B 0,C 180,E1 -16264.137,E2 -16264.137} C_VEL
LIN {X 0,Y 304.71,Z 823.726,A -85,B 0,C 180,E1 -16265.297,E2 -16265.297} C_VEL
LIN {X 0,Y 305.201,Z 836.184,A -85,B 0,C 180,E1 -16266.595,E2 -16266.595} C_VEL
LIN {X 0,Y 304.574,Z 849.045,A -85,B 0,C 180,E1 -16268.112,E2 -16268.112} C_VEL
LIN {X 0,Y 303.582,Z 861.172,A -85,B 0,C 180,E1 -16269.857,E2 -16269.857} C_VEL
LIN {X 0,Y 302.989,Z 866.285,A -85,B 0,C 180,E1 -16270.698,E2 -16270.698} C_VEL
LIN {X 0,Y 301.126,Z 875.206,A -85,B 0,C 180,E1 -16272.337,E2 -16272.337} C_VEL
LIN {X 0,Y 299.802,Z 882.576,A -85,B 0,C 180,E1 -16273.972,E2 -16273.972} C_VEL
LIN {X 0,Y 298.589,Z 890.353,A -85,B 0,C 180,E1 -16276.039,E2 -16276.039} C_VEL
LIN {X 0,Y 297.711,Z 897.479,A -85,B 0,C 180,E1 -16278.424,E2 -16278.424} C_VEL
LIN {X 0,Y 297.363,Z 902.343,A -85,B 0,C 180,E1 -16280.477,E2 -16280.477} C_VEL
LIN {X 0,Y 297.377,Z 906.929,A -85,B 0,C 180,E1 -16283.026,E2 -16283.026} C_VEL
LIN {X 0,Y 297.521,Z 908.96,A -85,B 0,C 180,E1 -16284.578,E2 -16284.578} C_VEL
LIN {X 0,Y 297.785,Z 910.3,A -85,B 0,C 180,E1 -16285.94,E2 -16285.94} C_VEL
LIN {X 0,Y 297.868,Z 911.199,A -85,B 0,C 180,E1 -16287.295,E2 -16287.295} C_VEL
LIN {X 0,Y 297.997,Z 911.68,A -85,B 0,C 180,E1 -16288.648,E2 -16288.648} C_VEL
LIN {X 0,Y 298.225,Z 911.708,A -85,B 0,C 180,E1 -16290,E2 -16290} C_VEL
LIN {X 0,Y 298.062,Z 911.252,A -85,B 0,C 180,E1 -16291.351,E2 -16291.351} C_VEL
LIN {X 0,Y 297.961,Z 910.386,A -85,B 0,C 180,E1 -16292.704,E2 -16292.704} C_VEL
LIN {X 0,Y 297.863,Z 909.07,A -85,B 0,C 180,E1 -16294.059,E2 -16294.059} C_VEL
LIN {X 0,Y 297.673,Z 906.184,A -85,B 0,C 180,E1 -16296.099,E2 -16296.099} C_VEL
LIN {X 0,Y 297.557,Z 902.171,A -85,B 0,C 180,E1 -16298.147,E2 -16298.147} C_VEL
LIN {X 0,Y 297.738,Z 895.932,A -85,B 0,C 180,E1 -16300.541,E2 -16300.541} C_VEL
LIN {X 0,Y 298.22,Z 889.118,A -85,B 0,C 180,E1 -16302.591,E2 -16302.591} C_VEL
LIN {X 0,Y 299.045,Z 880.624,A -85,B 0,C 180,E1 -16304.634,E2 -16304.634} C_VEL
LIN {X 0,Y 300.089,Z 871.941,A -85,B 0,C 180,E1 -16306.322,E2 -16306.322} C_VEL
LIN {X 0,Y 301.461,Z 861.359,A -85,B 0,C 180,E1 -16307.993,E2 -16307.993} C_VEL
LIN {X 0,Y 301.537,Z 854.858,A -85,B 0,C 180,E1 -16308.868,E2 -16308.868} C_VEL
LIN {X 0,Y 301.229,Z 842.162,A -85,B 0,C 180,E1 -16310.307,E2 -16310.307} C_VEL
LIN {X 0,Y 300.662,Z 829.836,A -85,B 0,C 180,E1 -16311.415,E2 -16311.415} C_VEL
LIN {X 0,Y 299.582,Z 815.705,A -85,B 0,C 180,E1 -16312.382,E2 -16312.382} C_VEL
LIN {X 0,Y 298.411,Z 803.339,A -85,B 0,C 180,E1 -16313.025,E2 -16313.025} C_VEL
LIN {X 0,Y 299.487,Z 792.217,A -85,B 0,C 180,E1 -16317.35,E2 -16317.35} C_VEL
LIN {X 0,Y 300.83,Z 781.136,A -85,B 0,C 180,E1 -16321.712,E2 -16321.712} C_VEL
LIN {X 0,Y 302.338,Z 771.517,A -85,B 0,C 180,E1 -16325.551,E2 -16325.551} C_VEL
LIN {X 0,Y 303.306,Z 765.416,A -85,B 0,C 180,E1 -16328.017,E2 -16328.017} C_VEL
LIN {X 0,Y 302.711,Z 760.86,A -85,B 0,C 180,E1 -16329.99,E2 -16329.99} C_VEL
LIN {X 0,Y 301.091,Z 752.776,A -85,B 0,C 180,E1 -16333.648,E2 -16333.648} C_VEL
LIN {X 0,Y 299.618,Z 745.456,A -85,B 0,C 180,E1 -16337.138,E2 -16337.138} C_VEL
LIN {X 0,Y 298.417,Z 739.314,A -85,B 0,C 180,E1 -16340.296,E2 -16340.296} C_VEL
LIN {X 0,Y 298.42,Z 739.312,A -85,B 0,C 180,E1 -16343.93,E2 -16343.93} C_VEL
LIN {X 0,Y 298.397,Z 739.316,A -85,B 0,C 180,E1 -16347.983,E2 -16347.983} C_VEL
LIN {X 0,Y 298.465,Z 739.309,A -85,B 0,C 180,E1 -16351.904,E2 -16351.904} C_VEL
LIN {X 0,Y 298.486,Z 739.301,A -85,B 0,C 180,E1 -16354.924,E2 -16354.924} C_VEL
LIN {X 0,Y 298.443,Z 739.306,A -85,B 0,C 180,E1 -16359.315,E2 -16359.315} C_VEL
LIN {X 0,Y 298.539,Z 739.299,A -85,B 0,C 180,E1 -16362.18,E2 -16362.18} C_VEL
LIN {X 0,Y 298.595,Z 739.288,A -85,B 0,C 180,E1 -16364.995,E2 -16364.995} C_VEL
LIN {X 0,Y 298.593,Z 739.287,A -85,B 0,C 180,E1 -16369.147,E2 -16369.147} C_VEL
LIN {X 0,Y 298.743,Z 739.27,A -85,B 0,C 180,E1 -16371.886,E2 -16371.886} C_VEL
LIN {X 0,Y 298.653,Z 739.285,A -85,B 0,C 180,E1 -16374.599,E2 -16374.599} C_VEL
LIN {X 0,Y 298.92,Z 739.252,A -85,B 0,C 180,E1 -16378.653,E2 -16378.653} C_VEL
LIN {X 0,Y 298.92,Z 739.247,A -85,B 0,C 180,E1 -16381.347,E2 -16381.347} C_VEL
LIN {X 0,Y 298.641,Z 739.282,A -85,B 0,C 180,E1 -16385.402,E2 -16385.402} C_VEL
LIN {X 0,Y 298.704,Z 739.273,A -85,B 0,C 180,E1 -16388.116,E2 -16388.116} C_VEL
LIN {X 0,Y 298.552,Z 739.293,A -85,B 0,C 180,E1 -16392.232,E2 -16392.232} C_VEL
LIN {X 0,Y 298.55,Z 739.297,A -85,B 0,C 180,E1 -16395.169,E2 -16395.169} C_VEL
LIN {X 0,Y 298.505,Z 739.304,A -85,B 0,C 180,E1 -16399.246,E2 -16399.246} C_VEL
LIN {X 0,Y 298.384,Z 739.316,A -85,B 0,C 180,E1 -16403.604,E2 -16403.604} C_VEL
LIN {X 0,Y 298.404,Z 739.311,A -85,B 0,C 180,E1 -16406.583,E2 -16406.583} C_VEL
LIN {X 0,Y 298.395,Z 739.317,A -85,B 0,C 180,E1 -16409.644,E2 -16409.644} C_VEL
LIN {X 0,Y 298.394,Z 739.312,A -85,B 0,C 180,E1 -16412.801,E2 -16412.801} C_VEL
LIN {X 0,Y 298.427,Z 739.308,A -85,B 0,C 180,E1 -16416.802,E2 -16416.802} C_VEL
LIN {X 0,Y 298.348,Z 739.319,A -85,B 0,C 180,E1 -16421.268,E2 -16421.268} C_VEL
LIN {X 0,Y 298.356,Z 739.317,A -85,B 0,C 180,E1 -16425.035,E2 -16425.035} C_VEL
LIN {X 0,Y 298.349,Z 739.318,A -85,B 0,C 180,E1 -16428.921,E2 -16428.921} C_VEL
LIN {X 0,Y 298.427,Z 739.308,A -85,B 0,C 180,E1 -16433.198,E2 -16433.198} C_VEL
LIN {X 0,Y 298.394,Z 739.312,A -85,B 0,C 180,E1 -16437.2,E2 -16437.2} C_VEL
LIN {X 0,Y 298.366,Z 739.319,A -85,B 0,C 180,E1 -16440.638,E2 -16440.638} C_VEL
LIN {X 0,Y 298.415,Z 739.312,A -85,B 0,C 180,E1 -16444.918,E2 -16444.918} C_VEL
LIN {X 0,Y 298.428,Z 739.308,A -85,B 0,C 180,E1 -16449.314,E2 -16449.314} C_VEL
LIN {X 0,Y 298.48,Z 739.303,A -85,B 0,C 180,E1 -16452.176,E2 -16452.176} C_VEL
LIN {X 0,Y 298.588,Z 739.291,A -85,B 0,C 180,E1 -16454.995,E2 -16454.995} C_VEL
LIN {X 0,Y 298.584,Z 739.292,A -85,B 0,C 180,E1 -16459.146,E2 -16459.146} C_VEL
LIN {X 0,Y 298.7,Z 739.274,A -85,B 0,C 180,E1 -16461.884,E2 -16461.884} C_VEL
LIN {X 0,Y 298.628,Z 739.285,A -85,B 0,C 180,E1 -16464.598,E2 -16464.598} C_VEL
LIN {X 0,Y 298.912,Z 739.249,A -85,B 0,C 180,E1 -16468.653,E2 -16468.653} C_VEL
LIN {X 0,Y 298.906,Z 739.253,A -85,B 0,C 180,E1 -16471.347,E2 -16471.347} C_VEL
LIN {X 0,Y 298.738,Z 739.27,A -85,B 0,C 180,E1 -16476.755,E2 -16476.755} C_VEL
LIN {X 0,Y 298.629,Z 739.288,A -85,B 0,C 180,E1 -16479.482,E2 -16479.482} C_VEL
LIN {X 0,Y 298.556,Z 739.297,A -85,B 0,C 180,E1 -16483.615,E2 -16483.615} C_VEL
LIN {X 0,Y 298.552,Z 739.293,A -85,B 0,C 180,E1 -16486.409,E2 -16486.409} C_VEL
LIN {X 0,Y 298.5,Z 739.304,A -85,B 0,C 180,E1 -16489.647,E2 -16489.647} C_VEL
LIN {X 0,Y 298.425,Z 739.312,A -85,B 0,C 180,E1 -16493.601,E2 -16493.601} C_VEL
LIN {X 0,Y 298.411,Z 739.311,A -85,B 0,C 180,E1 -16496.582,E2 -16496.582} C_VEL
LIN {X 0,Y 298.396,Z 739.315,A -85,B 0,C 180,E1 -16499.644,E2 -16499.644} C_VEL
LIN {X 0,Y 298.395,Z 739.313,A -85,B 0,C 180,E1 -16502.801,E2 -16502.801} C_VEL
LIN {X 0,Y 298.449,Z 739.307,A -85,B 0,C 180,E1 -16506.808,E2 -16506.808} C_VEL
LIN {X 0,Y 298.434,Z 739.314,A -85,B 0,C 180,E1 -16510.748,E2 -16510.748} C_VEL
LIN {X 0,Y 301.984,Z 751.189,A -85,B 0,C 180,E1 -16511.953,E2 -16511.953} C_VEL
LIN {X 0,Y 304.923,Z 762.245,A -85,B 0,C 180,E1 -16513.29,E2 -16513.29} C_VEL
LIN {X 0,Y 304.884,Z 766.043,A -85,B 0,C 180,E1 -16513.753,E2 -16513.753} C_VEL
LIN {X 0,Y 303.85,Z 776.971,A -85,B 0,C 180,E1 -16515.226,E2 -16515.226} C_VEL
LIN {X 0,Y 302.709,Z 787.575,A -85,B 0,C 180,E1 -16516.999,E2 -16516.999} C_VEL
LIN {X 0,Y 301.702,Z 796.641,A -85,B 0,C 180,E1 -16518.871,E2 -16518.871} C_VEL
LIN {X 0,Y 300.774,Z 804.505,A -85,B 0,C 180,E1 -16520.884,E2 -16520.884} C_VEL
LIN {X 0,Y 300.092,Z 810.52,A -85,B 0,C 180,E1 -16522.775,E2 -16522.775} C_VEL
LIN {X 0,Y 299.52,Z 815.551,A -85,B 0,C 180,E1 -16524.732,E2 -16524.732} C_VEL
LIN {X 0,Y 299.125,Z 820.534,A -85,B 0,C 180,E1 -16527.29,E2 -16527.29} C_VEL
LIN {X 0,Y 298.964,Z 822.748,A -85,B 0,C 180,E1 -16528.857,E2 -16528.857} C_VEL
LIN {X 0,Y 298.896,Z 824.455,A -85,B 0,C 180,E1 -16530.458,E2 -16530.458} C_VEL
LIN {X 0,Y 298.955,Z 825.495,A -85,B 0,C 180,E1 -16531.954,E2 -16531.954} C_VEL
LIN {X 0,Y 299.131,Z 826.091,A -85,B 0,C 180,E1 -16533.487,E2 -16533.487} C_VEL
LIN {X 0,Y 299.662,Z 825.818,A -85,B 0,C 180,E1 -16536.16,E2 -16536.16} C_VEL
LIN {X 0,Y 300.301,Z 824.713,A -85,B 0,C 180,E1 -16538.009,E2 -16538.009} C_VEL
LIN {X 0,Y 300.896,Z 823.258,A -85,B 0,C 180,E1 -16539.491,E2 -16539.491} C_VEL
LIN {X 0,Y 301.87,Z 820.162,A -85,B 0,C 180,E1 -16541.682,E2 -16541.682} C_VEL
LIN {X 0,Y 303.2,Z 815.825,A -85,B 0,C 180,E1 -16543.85,E2 -16543.85} C_VEL
LIN {X 0,Y 304.983,Z 809.442,A -85,B 0,C 180,E1 -16546.204,E2 -16546.204} C_VEL
LIN {X 0,Y 306.62,Z 802.887,A -85,B 0,C 180,E1 -16548.095,E2 -16548.095} C_VEL
LIN {X 0,Y 308.307,Z 795.464,A -85,B 0,C 180,E1 -16549.824,E2 -16549.824} C_VEL
LIN {X 0,Y 310.266,Z 785.411,A -85,B 0,C 180,E1 -16551.697,E2 -16551.697} C_VEL
LIN {X 0,Y 312.058,Z 775.281,A -85,B 0,C 180,E1 -16553.21,E2 -16553.21} C_VEL
LIN {X 0,Y 312.026,Z 773.129,A -85,B 0,C 180,E1 -16553.534,E2 -16553.534} C_VEL
LIN {X 0,Y 309.974,Z 765.367,A -85,B 0,C 180,E1 -16554.871,E2 -16554.871} C_VEL
LIN {X 0,Y 308.05,Z 761.47,A -85,B 0,C 180,E1 -16555.608,E2 -16555.608} C_VEL
LIN {X 0,Y 303.337,Z 756.117,A -85,B 0,C 180,E1 -16556.889,E2 -16556.889} C_VEL
LIN {X 0,Y 297.205,Z 749.857,A -85,B 0,C 180,E1 -16558.455,E2 -16558.455} C_VEL
LIN {X 0,Y 295.454,Z 747.403,A -85,B 0,C 180,E1 -16558.961,E2 -16558.961} C_VEL
LIN {X 0,Y 293.568,Z 743.862,A -85,B 0,C 180,E1 -16559.571,E2 -16559.571} C_VEL
LIN {X 0,Y 292.208,Z 741.366,A -85,B 0,C 180,E1 -16560,E2 -16560} C_VEL
LIN {X 0,Y 291.933,Z 740.121,A -85,B 0,C 180,E1 -16560.172,E2 -16560.172} C_VEL
LIN {X 0,Y 291.788,Z 740.131,A -85,B 0,C 180,E1 -16562.761,E2 -16562.761} C_VEL
LIN {X 0,Y 291.738,Z 740.142,A -85,B 0,C 180,E1 -16566.918,E2 -16566.918} C_VEL
LIN {X 0,Y 291.578,Z 740.158,A -85,B 0,C 180,E1 -16569.713,E2 -16569.713} C_VEL
LIN {X 0,Y 291.525,Z 740.17,A -85,B 0,C 180,E1 -16573.95,E2 -16573.95} C_VEL
LIN {X 0,Y 291.49,Z 740.177,A -85,B 0,C 180,E1 -16576.818,E2 -16576.818} C_VEL
LIN {X 0,Y 291.453,Z 740.181,A -85,B 0,C 180,E1 -16579.875,E2 -16579.875} C_VEL
LIN {X 0,Y 291.384,Z 740.183,A -85,B 0,C 180,E1 -16584.207,E2 -16584.207} C_VEL
LIN {X 0,Y 291.421,Z 740.183,A -85,B 0,C 180,E1 -16587.272,E2 -16587.272} C_VEL
LIN {X 0,Y 291.344,Z 740.191,A -85,B 0,C 180,E1 -16591.443,E2 -16591.443} C_VEL
LIN {X 0,Y 292.139,Z 743.728,A -85,B 0,C 180,E1 -16595.266,E2 -16595.266} C_VEL
LIN {X 0,Y 293.034,Z 747.49,A -85,B 0,C 180,E1 -16598.578,E2 -16598.578} C_VEL
LIN {X 0,Y 294.023,Z 752.303,A -85,B 0,C 180,E1 -16602.184,E2 -16602.184} C_VEL
LIN {X 0,Y 295.083,Z 757.56,A -85,B 0,C 180,E1 -16605.603,E2 -16605.603} C_VEL
LIN {X 0,Y 296.3,Z 764.125,A -85,B 0,C 180,E1 -16609.378,E2 -16609.378} C_VEL
LIN {X 0,Y 296.685,Z 768.068,A -85,B 0,C 180,E1 -16611.418,E2 -16611.418} C_VEL
LIN {X 0,Y 295.381,Z 774.916,A -85,B 0,C 180,E1 -16614.538,E2 -16614.538} C_VEL
LIN {X 0,Y 293.365,Z 786.696,A -85,B 0,C 180,E1 -16619.591,E2 -16619.591} C_VEL
LIN {X 0,Y 292.721,Z 791.698,A -85,B 0,C 180,E1 -16621.586,E2 -16621.586} C_VEL
LIN {X 0,Y 293.705,Z 795.7,A -85,B 0,C 180,E1 -16621.929,E2 -16621.929} C_VEL
LIN {X 0,Y 296.501,Z 808.997,A -85,B 0,C 180,E1 -16623.142,E2 -16623.142} C_VEL
LIN {X 0,Y 298.144,Z 821.569,A -85,B 0,C 180,E1 -16624.386,E2 -16624.386} C_VEL
LIN {X 0,Y 298.745,Z 835.374,A -85,B 0,C 180,E1 -16625.873,E2 -16625.873} C_VEL
LIN {X 0,Y 298.122,Z 847.841,A -85,B 0,C 180,E1 -16627.406,E2 -16627.406} C_VEL
LIN {X 0,Y 296.913,Z 860.009,A -85,B 0,C 180,E1 -16629.203,E2 -16629.203} C_VEL
LIN {X 0,Y 296.281,Z 866.111,A -85,B 0,C 180,E1 -16630.243,E2 -16630.243} C_VEL
LIN {X 0,Y 294.013,Z 876.407,A -85,B 0,C 180,E1 -16632.255,E2 -16632.255} C_VEL
LIN {X 0,Y 292.317,Z 884.701,A -85,B 0,C 180,E1 -16634.257,E2 -16634.257} C_VEL
LIN {X 0,Y 291.657,Z 889.699,A -85,B 0,C 180,E1 -16635.7,E2 -16635.7} C_VEL
LIN {X 0,Y 290.701,Z 896.724,A -85,B 0,C 180,E1 -16638.141,E2 -16638.141} C_VEL
LIN {X 0,Y 290.305,Z 901.514,A -85,B 0,C 180,E1 -16640.243,E2 -16640.243} C_VEL
LIN {X 0,Y 290.255,Z 905.357,A -85,B 0,C 180,E1 -16642.417,E2 -16642.417} C_VEL
LIN {X 0,Y 290.435,Z 907.999,A -85,B 0,C 180,E1 -16644.445,E2 -16644.445} C_VEL
LIN {X 0,Y 290.7,Z 909.309,A -85,B 0,C 180,E1 -16645.841,E2 -16645.841} C_VEL
LIN {X 0,Y 290.822,Z 910.189,A -85,B 0,C 180,E1 -16647.23,E2 -16647.23} C_VEL
LIN {X 0,Y 290.965,Z 910.619,A -85,B 0,C 180,E1 -16648.616,E2 -16648.616} C_VEL
LIN {X 0,Y 291.213,Z 910.621,A -85,B 0,C 180,E1 -16650,E2 -16650} C_VEL
LIN {X 0,Y 291.036,Z 910.138,A -85,B 0,C 180,E1 -16651.384,E2 -16651.384} C_VEL
LIN {X 0,Y 290.927,Z 909.24,A -85,B 0,C 180,E1 -16652.769,E2 -16652.769} C_VEL
LIN {X 0,Y 290.825,Z 907.858,A -85,B 0,C 180,E1 -16654.157,E2 -16654.157} C_VEL
LIN {X 0,Y 290.623,Z 904.905,A -85,B 0,C 180,E1 -16656.247,E2 -16656.247} C_VEL
LIN {X 0,Y 290.505,Z 900.814,A -85,B 0,C 180,E1 -16658.346,E2 -16658.346} C_VEL
LIN {X 0,Y 290.697,Z 894.492,A -85,B 0,C 180,E1 -16660.799,E2 -16660.799} C_VEL
LIN {X 0,Y 291.21,Z 887.586,A -85,B 0,C 180,E1 -16662.899,E2 -16662.899} C_VEL
LIN {X 0,Y 291.939,Z 880.54,A -85,B 0,C 180,E1 -16664.642,E2 -16664.642} C_VEL
LIN {X 0,Y 293.085,Z 871.184,A -85,B 0,C 180,E1 -16666.528,E2 -16666.528} C_VEL
LIN {X 0,Y 294.343,Z 861.702,A -85,B 0,C 180,E1 -16668.083,E2 -16668.083} C_VEL
LIN {X 0,Y 294.562,Z 856.761,A -85,B 0,C 180,E1 -16668.79,E2 -16668.79} C_VEL
LIN {X 0,Y 294.317,Z 844.949,A -85,B 0,C 180,E1 -16670.258,E2 -16670.258} C_VEL
LIN {X 0,Y 293.846,Z 832.506,A -85,B 0,C 180,E1 -16671.483,E2 -16671.483} C_VEL
LIN {X 0,Y 292.923,Z 819.675,A -85,B 0,C 180,E1 -16672.481,E2 -16672.481} C_VEL
LIN {X 0,Y 291.754,Z 806.31,A -85,B 0,C 180,E1 -16673.243,E2 -16673.243} C_VEL
LIN {X 0,Y 291.409,Z 802.387,A -85,B 0,C 180,E1 -16673.441,E2 -16673.441} C_VEL
LIN {X 0,Y 292.56,Z 791.189,A -85,B 0,C 180,E1 -16677.932,E2 -16677.932} C_VEL
LIN {X 0,Y 294.056,Z 779.841,A -85,B 0,C 180,E1 -16682.531,E2 -16682.531} C_VEL
LIN {X 0,Y 295.643,Z 770.249,A -85,B 0,C 180,E1 -16686.463,E2 -16686.463} C_VEL
LIN {X 0,Y 296.227,Z 765.476,A -85,B 0,C 180,E1 -16688.47,E2 -16688.47} C_VEL
LIN {X 0,Y 295.18,Z 759.336,A -85,B 0,C 180,E1 -16691.232,E2 -16691.232} C_VEL
LIN {X 0,Y 293.535,Z 751.216,A -85,B 0,C 180,E1 -16695.065,E2 -16695.065} C_VEL
LIN {X 0,Y 291.846,Z 742.436,A -85,B 0,C 180,E1 -16699.444,E2 -16699.444} C_VEL
LIN {X 0,Y 291.384,Z 740.189,A -85,B 0,C 180,E1 -16700.636,E2 -16700.636} C_VEL
LIN {X 0,Y 291.408,Z 740.183,A -85,B 0,C 180,E1 -16702.92,E2 -16702.92} C_VEL
